LIN {X 0,Y 566.232,Z 349.956,A -85,B 0,C 180,E1 -2396.899,E2 -2396.899} C_VEL
LIN {X 0,Y 566.183,Z 349.956,A -85,B 0,C 180,E1 -2399.407,E2 -2399.407} C_VEL
LIN {X 0,Y 566.232,Z 349.955,A -85,B 0,C 180,E1 -2401.859,E2 -2401.859} C_VEL
LIN {X 0,Y 566.218,Z 349.953,A -85,B 0,C 180,E1 -2404.251,E2 -2404.251} C_VEL
LIN {X 0,Y 566.176,Z 349.96,A -85,B 0,C 180,E1 -2406.718,E2 -2406.718} C_VEL
LIN {X 0,Y 566.215,Z 349.952,A -85,B 0,C 180,E1 -2409.663,E2 -2409.663} C_VEL
LIN {X 0,Y 566.207,Z 349.954,A -85,B 0,C 180,E1 -2412.669,E2 -2412.669} C_VEL
LIN {X 0,Y 566.238,Z 349.953,A -85,B 0,C 180,E1 -2415.627,E2 -2415.627} C_VEL
LIN {X 0,Y 566.239,Z 349.956,A -85,B 0,C 180,E1 -2418.675,E2 -2418.675} C_VEL
LIN {X 0,Y 566.23,Z 349.95,A -85,B 0,C 180,E1 -2421.434,E2 -2421.434} C_VEL
LIN {X 0,Y 566.266,Z 349.947,A -85,B 0,C 180,E1 -2424.302,E2 -2424.302} C_VEL
LIN {X 0,Y 566.287,Z 349.944,A -85,B 0,C 180,E1 -2427.866,E2 -2427.866} C_VEL
LIN {X 0,Y 566.306,Z 349.944,A -85,B 0,C 180,E1 -2430.711,E2 -2430.711} C_VEL
LIN {X 0,Y 566.272,Z 349.945,A -85,B 0,C 180,E1 -2432.846,E2 -2432.846} C_VEL
LIN {X 0,Y 566.268,Z 349.949,A -85,B 0,C 180,E1 -2435.698,E2 -2435.698} C_VEL
LIN {X 0,Y 566.231,Z 349.955,A -85,B 0,C 180,E1 -2438.566,E2 -2438.566} C_VEL
LIN {X 0,Y 566.246,Z 349.949,A -85,B 0,C 180,E1 -2441.454,E2 -2441.454} C_VEL
LIN {X 0,Y 566.238,Z 349.949,A -85,B 0,C 180,E1 -2444.507,E2 -2444.507} C_VEL
LIN {X 0,Y 566.204,Z 349.958,A -85,B 0,C 180,E1 -2447.332,E2 -2447.332} C_VEL
LIN {X 0,Y 566.213,Z 349.959,A -85,B 0,C 180,E1 -2450.337,E2 -2450.337} C_VEL
LIN {X 0,Y 566.177,Z 349.958,A -85,B 0,C 180,E1 -2453.282,E2 -2453.282} C_VEL
LIN {X 0,Y 566.218,Z 349.955,A -85,B 0,C 180,E1 -2455.749,E2 -2455.749} C_VEL
LIN {X 0,Y 566.207,Z 349.954,A -85,B 0,C 180,E1 -2458.202,E2 -2458.202} C_VEL
LIN {X 0,Y 566.194,Z 349.956,A -85,B 0,C 180,E1 -2461.076,E2 -2461.076} C_VEL
LIN {X 0,Y 566.215,Z 349.959,A -85,B 0,C 180,E1 -2463.734,E2 -2463.734} C_VEL
LIN {X 0,Y 566.203,Z 349.954,A -85,B 0,C 180,E1 -2466.57,E2 -2466.57} C_VEL
LIN {X 0,Y 566.219,Z 349.952,A -85,B 0,C 180,E1 -2469.686,E2 -2469.686} C_VEL
LIN {X 0,Y 566.218,Z 349.958,A -85,B 0,C 180,E1 -2472.087,E2 -2472.087} C_VEL
LIN {X 0,Y 566.172,Z 349.959,A -85,B 0,C 180,E1 -2475.036,E2 -2475.036} C_VEL
LIN {X 0,Y 566.192,Z 349.955,A -85,B 0,C 180,E1 -2477.91,E2 -2477.91} C_VEL
LIN {X 0,Y 566.226,Z 349.955,A -85,B 0,C 180,E1 -2480.727,E2 -2480.727} C_VEL
LIN {X 0,Y 566.211,Z 349.959,A -85,B 0,C 180,E1 -2483.785,E2 -2483.785} C_VEL
LIN {X 0,Y 566.216,Z 349.952,A -85,B 0,C 180,E1 -2486.266,E2 -2486.266} C_VEL
LIN {X 0,Y 566.198,Z 349.961,A -85,B 0,C 180,E1 -2488.923,E2 -2488.923} C_VEL
LIN {X 0,Y 566.253,Z 350.125,A -85,B 0,C 180,E1 -2490.234,E2 -2490.234} C_VEL
LIN {X 0,Y 566.179,Z 357.411,A -85,B 0,C 180,E1 -2493.347,E2 -2493.347} C_VEL
LIN {X 0,Y 566.127,Z 363.027,A -85,B 0,C 180,E1 -2495.816,E2 -2495.816} C_VEL
LIN {X 0,Y 566.063,Z 370.064,A -85,B 0,C 180,E1 -2498.897,E2 -2498.897} C_VEL
LIN {X 0,Y 566.005,Z 377.154,A -85,B 0,C 180,E1 -2501.915,E2 -2501.915} C_VEL
LIN {X 0,Y 565.961,Z 382.566,A -85,B 0,C 180,E1 -2504.146,E2 -2504.146} C_VEL
LIN {X 0,Y 565.962,Z 387.979,A -85,B 0,C 180,E1 -2506.353,E2 -2506.353} C_VEL
LIN {X 0,Y 565.925,Z 395.195,A -85,B 0,C 180,E1 -2509.264,E2 -2509.264} C_VEL
LIN {X 0,Y 565.928,Z 403.709,A -85,B 0,C 180,E1 -2512.665,E2 -2512.665} C_VEL
LIN {X 0,Y 566.231,Z 412.154,A -85,B 0,C 180,E1 -2512.959,E2 -2512.959} C_VEL
LIN {X 0,Y 566.146,Z 420.811,A -85,B 0,C 180,E1 -2513.393,E2 -2513.393} C_VEL
LIN {X 0,Y 566.094,Z 429.047,A -85,B 0,C 180,E1 -2513.942,E2 -2513.942} C_VEL
LIN {X 0,Y 566.027,Z 437.057,A -85,B 0,C 180,E1 -2514.657,E2 -2514.657} C_VEL
LIN {X 0,Y 566.028,Z 443.23,A -85,B 0,C 180,E1 -2515.371,E2 -2515.371} C_VEL
LIN {X 0,Y 566.012,Z 448.087,A -85,B 0,C 180,E1 -2516.084,E2 -2516.084} C_VEL
LIN {X 0,Y 565.934,Z 451.834,A -85,B 0,C 180,E1 -2516.796,E2 -2516.796} C_VEL
LIN {X 0,Y 565.855,Z 455.839,A -85,B 0,C 180,E1 -2517.865,E2 -2517.865} C_VEL
LIN {X 0,Y 565.848,Z 457.579,A -85,B 0,C 180,E1 -2518.577,E2 -2518.577} C_VEL
LIN {X 0,Y 565.842,Z 458.621,A -85,B 0,C 180,E1 -2519.288,E2 -2519.288} C_VEL
LIN {X 0,Y 565.839,Z 458.996,A -85,B 0,C 180,E1 -2520,E2 -2520} C_VEL
LIN {X 0,Y 565.841,Z 458.711,A -85,B 0,C 180,E1 -2520.712,E2 -2520.712} C_VEL
LIN {X 0,Y 565.848,Z 457.761,A -85,B 0,C 180,E1 -2521.423,E2 -2521.423} C_VEL
LIN {X 0,Y 565.854,Z 456.12,A -85,B 0,C 180,E1 -2522.135,E2 -2522.135} C_VEL
LIN {X 0,Y 565.893,Z 453.732,A -85,B 0,C 180,E1 -2522.847,E2 -2522.847} C_VEL
LIN {X 0,Y 565.991,Z 448.601,A -85,B 0,C 180,E1 -2523.916,E2 -2523.916} C_VEL
LIN {X 0,Y 566.035,Z 442.528,A -85,B 0,C 180,E1 -2524.808,E2 -2524.808} C_VEL
LIN {X 0,Y 565.983,Z 436.212,A -85,B 0,C 180,E1 -2525.522,E2 -2525.522} C_VEL
LIN {X 0,Y 566.114,Z 429.057,A -85,B 0,C 180,E1 -2526.147,E2 -2526.147} C_VEL
LIN {X 0,Y 566.115,Z 420.691,A -85,B 0,C 180,E1 -2526.705,E2 -2526.705} C_VEL
LIN {X 0,Y 566.246,Z 411.008,A -85,B 0,C 180,E1 -2527.174,E2 -2527.174} C_VEL
LIN {X 0,Y 565.909,Z 403.653,A -85,B 0,C 180,E1 -2527.448,E2 -2527.448} C_VEL
LIN {X 0,Y 565.924,Z 395.42,A -85,B 0,C 180,E1 -2530.736,E2 -2530.736} C_VEL
LIN {X 0,Y 565.943,Z 388.201,A -85,B 0,C 180,E1 -2533.647,E2 -2533.647} C_VEL
LIN {X 0,Y 565.976,Z 380.981,A -85,B 0,C 180,E1 -2536.595,E2 -2536.595} C_VEL
LIN {X 0,Y 566.022,Z 374.496,A -85,B 0,C 180,E1 -2539.325,E2 -2539.325} C_VEL
LIN {X 0,Y 566.094,Z 368.863,A -85,B 0,C 180,E1 -2541.867,E2 -2541.867} C_VEL
LIN {X 0,Y 566.164,Z 363.641,A -85,B 0,C 180,E1 -2544.182,E2 -2544.182} C_VEL
LIN {X 0,Y 566.204,Z 357.666,A -85,B 0,C 180,E1 -2546.658,E2 -2546.658} C_VEL
LIN {X 0,Y 566.274,Z 349.951,A -85,B 0,C 180,E1 -2549.97,E2 -2549.97} C_VEL
LIN {X 0,Y 566.224,Z 349.956,A -85,B 0,C 180,E1 -2553.102,E2 -2553.102} C_VEL
LIN {X 0,Y 566.167,Z 349.964,A -85,B 0,C 180,E1 -2555.692,E2 -2555.692} C_VEL
LIN {X 0,Y 566.22,Z 349.956,A -85,B 0,C 180,E1 -2558.559,E2 -2558.559} C_VEL
LIN {X 0,Y 566.216,Z 349.959,A -85,B 0,C 180,E1 -2561.136,E2 -2561.136} C_VEL
LIN {X 0,Y 566.205,Z 349.959,A -85,B 0,C 180,E1 -2564.035,E2 -2564.035} C_VEL
LIN {X 0,Y 566.209,Z 349.958,A -85,B 0,C 180,E1 -2567.082,E2 -2567.082} C_VEL
LIN {X 0,Y 566.21,Z 349.958,A -85,B 0,C 180,E1 -2569.801,E2 -2569.801} C_VEL
LIN {X 0,Y 566.201,Z 349.961,A -85,B 0,C 180,E1 -2572.599,E2 -2572.599} C_VEL
LIN {X 0,Y 566.203,Z 349.959,A -85,B 0,C 180,E1 -2575.181,E2 -2575.181} C_VEL
LIN {X 0,Y 566.236,Z 349.957,A -85,B 0,C 180,E1 -2577.744,E2 -2577.744} C_VEL
LIN {X 0,Y 566.232,Z 350.075,A -85,B 0,C 180,E1 -2580.922,E2 -2580.922} C_VEL
LIN {X 0,Y 567.515,Z 356.097,A -85,B 0,C 180,E1 -2582.128,E2 -2582.128} C_VEL
LIN {X 0,Y 567.256,Z 368.377,A -85,B 0,C 180,E1 -2584.302,E2 -2584.302} C_VEL
LIN {X 0,Y 567.027,Z 381.516,A -85,B 0,C 180,E1 -2586.519,E2 -2586.519} C_VEL
LIN {X 0,Y 566.812,Z 397.208,A -85,B 0,C 180,E1 -2589.116,E2 -2589.116} C_VEL
LIN {X 0,Y 566.567,Z 414.516,A -85,B 0,C 180,E1 -2591.934,E2 -2591.934} C_VEL
LIN {X 0,Y 566.392,Z 432.979,A -85,B 0,C 180,E1 -2594.896,E2 -2594.896} C_VEL
LIN {X 0,Y 566.217,Z 447.98,A -85,B 0,C 180,E1 -2597.272,E2 -2597.272} C_VEL
LIN {X 0,Y 566.942,Z 453.599,A -85,B 0,C 180,E1 -2597.38,E2 -2597.38} C_VEL
LIN {X 0,Y 566.899,Z 466.689,A -85,B 0,C 180,E1 -2597.674,E2 -2597.674} C_VEL
LIN {X 0,Y 566.748,Z 479.914,A -85,B 0,C 180,E1 -2598.13,E2 -2598.13} C_VEL
LIN {X 0,Y 566.61,Z 492.108,A -85,B 0,C 180,E1 -2598.705,E2 -2598.705} C_VEL
LIN {X 0,Y 566.485,Z 502.907,A -85,B 0,C 180,E1 -2599.365,E2 -2599.365} C_VEL
LIN {X 0,Y 566.339,Z 513.539,A -85,B 0,C 180,E1 -2600.175,E2 -2600.175} C_VEL
LIN {X 0,Y 566.207,Z 523.111,A -85,B 0,C 180,E1 -2601.074,E2 -2601.074} C_VEL
LIN {X 0,Y 566.112,Z 530.959,A -85,B 0,C 180,E1 -2601.971,E2 -2601.971} C_VEL
LIN {X 0,Y 566.001,Z 538.621,A -85,B 0,C 180,E1 -2603.046,E2 -2603.046} C_VEL
LIN {X 0,Y 566.004,Z 545.679,A -85,B 0,C 180,E1 -2604.299,E2 -2604.299} C_VEL
LIN {X 0,Y 565.933,Z 550.372,A -85,B 0,C 180,E1 -2605.37,E2 -2605.37} C_VEL
LIN {X 0,Y 565.927,Z 553.957,A -85,B 0,C 180,E1 -2606.44,E2 -2606.44} C_VEL
LIN {X 0,Y 565.878,Z 555.808,A -85,B 0,C 180,E1 -2607.152,E2 -2607.152} C_VEL
LIN {X 0,Y 565.846,Z 558.185,A -85,B 0,C 180,E1 -2608.576,E2 -2608.576} C_VEL
LIN {X 0,Y 565.839,Z 559,A -85,B 0,C 180,E1 -2610,E2 -2610} C_VEL
LIN {X 0,Y 565.846,Z 558.186,A -85,B 0,C 180,E1 -2611.423,E2 -2611.423} C_VEL
LIN {X 0,Y 565.878,Z 555.81,A -85,B 0,C 180,E1 -2612.847,E2 -2612.847} C_VEL
LIN {X 0,Y 565.926,Z 552.897,A -85,B 0,C 180,E1 -2613.916,E2 -2613.916} C_VEL
LIN {X 0,Y 565.878,Z 548.95,A -85,B 0,C 180,E1 -2614.987,E2 -2614.987} C_VEL
LIN {X 0,Y 566.002,Z 543.868,A -85,B 0,C 180,E1 -2616.058,E2 -2616.058} C_VEL
LIN {X 0,Y 566.04,Z 537.468,A -85,B 0,C 180,E1 -2617.132,E2 -2617.132} C_VEL
LIN {X 0,Y 566.133,Z 529.48,A -85,B 0,C 180,E1 -2618.208,E2 -2618.208} C_VEL
LIN {X 0,Y 566.229,Z 521.336,A -85,B 0,C 180,E1 -2619.105,E2 -2619.105} C_VEL
LIN {X 0,Y 566.35,Z 511.402,A -85,B 0,C 180,E1 -2620.005,E2 -2620.005} C_VEL
LIN {X 0,Y 566.524,Z 500.284,A -85,B 0,C 180,E1 -2620.808,E2 -2620.808} C_VEL
LIN {X 0,Y 566.66,Z 489.178,A -85,B 0,C 180,E1 -2621.446,E2 -2621.446} C_VEL
LIN {X 0,Y 566.746,Z 476.986,A -85,B 0,C 180,E1 -2621.988,E2 -2621.988} C_VEL
LIN {X 0,Y 566.887,Z 464.18,A -85,B 0,C 180,E1 -2622.394,E2 -2622.394} C_VEL
LIN {X 0,Y 566.827,Z 452.111,A -85,B 0,C 180,E1 -2622.645,E2 -2622.645} C_VEL
LIN {X 0,Y 566.216,Z 447.982,A -85,B 0,C 180,E1 -2622.728,E2 -2622.728} C_VEL
LIN {X 0,Y 566.399,Z 431.827,A -85,B 0,C 180,E1 -2625.288,E2 -2625.288} C_VEL
LIN {X 0,Y 566.568,Z 414.518,A -85,B 0,C 180,E1 -2628.066,E2 -2628.066} C_VEL
LIN {X 0,Y 566.791,Z 398.363,A -85,B 0,C 180,E1 -2630.695,E2 -2630.695} C_VEL
LIN {X 0,Y 567.037,Z 381.524,A -85,B 0,C 180,E1 -2633.483,E2 -2633.483} C_VEL
LIN {X 0,Y 567.381,Z 363.879,A -85,B 0,C 180,E1 -2636.482,E2 -2636.482} C_VEL
LIN {X 0,Y 567.421,Z 355.866,A -85,B 0,C 180,E1 -2637.876,E2 -2637.876} C_VEL
LIN {X 0,Y 566.23,Z 349.956,A -85,B 0,C 180,E1 -2639.002,E2 -2639.002} C_VEL
LIN {X 0,Y 566.235,Z 349.953,A -85,B 0,C 180,E1 -2642.256,E2 -2642.256} C_VEL
LIN {X 0,Y 566.184,Z 349.962,A -85,B 0,C 180,E1 -2644.99,E2 -2644.99} C_VEL
LIN {X 0,Y 566.198,Z 349.955,A -85,B 0,C 180,E1 -2647.461,E2 -2647.461} C_VEL
LIN {X 0,Y 566.209,Z 349.96,A -85,B 0,C 180,E1 -2650.199,E2 -2650.199} C_VEL
LIN {X 0,Y 566.208,Z 349.955,A -85,B 0,C 180,E1 -2653.054,E2 -2653.054} C_VEL
LIN {X 0,Y 566.204,Z 349.954,A -85,B 0,C 180,E1 -2656.048,E2 -2656.048} C_VEL
LIN {X 0,Y 566.222,Z 349.951,A -85,B 0,C 180,E1 -2659.212,E2 -2659.212} C_VEL
LIN {X 0,Y 566.192,Z 349.959,A -85,B 0,C 180,E1 -2661.637,E2 -2661.637} C_VEL
LIN {X 0,Y 566.199,Z 349.955,A -85,B 0,C 180,E1 -2664.31,E2 -2664.31} C_VEL
LIN {X 0,Y 566.222,Z 349.957,A -85,B 0,C 180,E1 -2666.898,E2 -2666.898} C_VEL
LIN {X 0,Y 566.19,Z 349.955,A -85,B 0,C 180,E1 -2669.408,E2 -2669.408} C_VEL
LIN {X 0,Y 566.231,Z 349.957,A -85,B 0,C 180,E1 -2671.858,E2 -2671.858} C_VEL
LIN {X 0,Y 566.215,Z 349.953,A -85,B 0,C 180,E1 -2674.251,E2 -2674.251} C_VEL
LIN {X 0,Y 566.171,Z 349.963,A -85,B 0,C 180,E1 -2676.719,E2 -2676.719} C_VEL
LIN {X 0,Y 566.215,Z 349.953,A -85,B 0,C 180,E1 -2679.663,E2 -2679.663} C_VEL
LIN {X 0,Y 566.201,Z 349.954,A -85,B 0,C 180,E1 -2682.668,E2 -2682.668} C_VEL
LIN {X 0,Y 566.237,Z 349.952,A -85,B 0,C 180,E1 -2685.627,E2 -2685.627} C_VEL
LIN {X 0,Y 566.237,Z 349.955,A -85,B 0,C 180,E1 -2688.675,E2 -2688.675} C_VEL
LIN {X 0,Y 566.23,Z 349.952,A -85,B 0,C 180,E1 -2691.434,E2 -2691.434} C_VEL
LIN {X 0,Y 566.258,Z 349.947,A -85,B 0,C 180,E1 -2694.302,E2 -2694.302} C_VEL
LIN {X 0,Y 566.278,Z 349.945,A -85,B 0,C 180,E1 -2697.866,E2 -2697.866} C_VEL
LIN {X 0,Y 566.305,Z 349.943,A -85,B 0,C 180,E1 -2700.711,E2 -2700.711} C_VEL
LIN {X 0,Y 566.275,Z 349.945,A -85,B 0,C 180,E1 -2702.846,E2 -2702.846} C_VEL
LIN {X 0,Y 566.261,Z 349.948,A -85,B 0,C 180,E1 -2705.698,E2 -2705.698} C_VEL
LIN {X 0,Y 566.236,Z 349.956,A -85,B 0,C 180,E1 -2708.566,E2 -2708.566} C_VEL
LIN {X 0,Y 566.244,Z 349.95,A -85,B 0,C 180,E1 -2711.454,E2 -2711.454} C_VEL
LIN {X 0,Y 566.236,Z 349.949,A -85,B 0,C 180,E1 -2714.507,E2 -2714.507} C_VEL
LIN {X 0,Y 566.202,Z 349.956,A -85,B 0,C 180,E1 -2717.332,E2 -2717.332} C_VEL
LIN {X 0,Y 566.216,Z 349.959,A -85,B 0,C 180,E1 -2720.337,E2 -2720.337} C_VEL
LIN {X 0,Y 566.191,Z 349.96,A -85,B 0,C 180,E1 -2723.404,E2 -2723.404} C_VEL
LIN {X 0,Y 566.215,Z 349.953,A -85,B 0,C 180,E1 -2725.749,E2 -2725.749} C_VEL
LIN {X 0,Y 566.205,Z 349.954,A -85,B 0,C 180,E1 -2727.483,E2 -2727.483} C_VEL
LIN {X 0,Y 565.525,Z 350.04,A -85,B 0,C 180,E1 -2728.077,E2 -2728.077} C_VEL
LIN {X 0,Y 562.659,Z 350.397,A -85,B 0,C 180,E1 -2729.04,E2 -2729.04} C_VEL
LIN {X 0,Y 560.249,Z 350.699,A -85,B 0,C 180,E1 -2729.816,E2 -2729.816} C_VEL
LIN {X 0,Y 559.222,Z 350.829,A -85,B 0,C 180,E1 -2730.414,E2 -2730.414} C_VEL
LIN {X 0,Y 559.141,Z 350.835,A -85,B 0,C 180,E1 -2730.617,E2 -2730.617} C_VEL
LIN {X 0,Y 559.167,Z 350.837,A -85,B 0,C 180,E1 -2733.575,E2 -2733.575} C_VEL
LIN {X 0,Y 559.16,Z 350.832,A -85,B 0,C 180,E1 -2736.447,E2 -2736.447} C_VEL
LIN {X 0,Y 559.18,Z 350.832,A -85,B 0,C 180,E1 -2738.934,E2 -2738.934} C_VEL
LIN {X 0,Y 559.193,Z 350.831,A -85,B 0,C 180,E1 -2741.768,E2 -2741.768} C_VEL
LIN {X 0,Y 559.142,Z 350.834,A -85,B 0,C 180,E1 -2744.739,E2 -2744.739} C_VEL
LIN {X 0,Y 559.167,Z 350.833,A -85,B 0,C 180,E1 -2747.257,E2 -2747.257} C_VEL
LIN {X 0,Y 559.182,Z 350.832,A -85,B 0,C 180,E1 -2750.135,E2 -2750.135} C_VEL
LIN {X 0,Y 559.143,Z 350.834,A -85,B 0,C 180,E1 -2752.892,E2 -2752.892} C_VEL
LIN {X 0,Y 559.169,Z 350.831,A -85,B 0,C 180,E1 -2756.051,E2 -2756.051} C_VEL
LIN {X 0,Y 559.158,Z 350.834,A -85,B 0,C 180,E1 -2758.981,E2 -2758.981} C_VEL
LIN {X 0,Y 559.173,Z 350.831,A -85,B 0,C 180,E1 -2761.619,E2 -2761.619} C_VEL
LIN {X 0,Y 559.185,Z 350.833,A -85,B 0,C 180,E1 -2763.903,E2 -2763.903} C_VEL
LIN {X 0,Y 559.145,Z 350.835,A -85,B 0,C 180,E1 -2766.571,E2 -2766.571} C_VEL
LIN {X 0,Y 559.182,Z 350.828,A -85,B 0,C 180,E1 -2769.396,E2 -2769.396} C_VEL
LIN {X 0,Y 559.154,Z 350.834,A -85,B 0,C 180,E1 -2771.686,E2 -2771.686} C_VEL
LIN {X 0,Y 559.171,Z 350.834,A -85,B 0,C 180,E1 -2773.948,E2 -2773.948} C_VEL
LIN {X 0,Y 559.176,Z 350.83,A -85,B 0,C 180,E1 -2776.184,E2 -2776.184} C_VEL
LIN {X 0,Y 559.199,Z 350.828,A -85,B 0,C 180,E1 -2779.134,E2 -2779.134} C_VEL
LIN {X 0,Y 559.207,Z 350.832,A -85,B 0,C 180,E1 -2782.054,E2 -2782.054} C_VEL
LIN {X 0,Y 559.26,Z 350.821,A -85,B 0,C 180,E1 -2784.954,E2 -2784.954} C_VEL
LIN {X 0,Y 559.258,Z 350.819,A -85,B 0,C 180,E1 -2787.84,E2 -2787.84} C_VEL
LIN {X 0,Y 559.276,Z 350.819,A -85,B 0,C 180,E1 -2790.72,E2 -2790.72} C_VEL
LIN {X 0,Y 559.239,Z 350.821,A -85,B 0,C 180,E1 -2792.882,E2 -2792.882} C_VEL
LIN {X 0,Y 559.236,Z 350.824,A -85,B 0,C 180,E1 -2795.77,E2 -2795.77} C_VEL
LIN {X 0,Y 559.19,Z 350.833,A -85,B 0,C 180,E1 -2798.674,E2 -2798.674} C_VEL
LIN {X 0,Y 559.209,Z 350.826,A -85,B 0,C 180,E1 -2801.601,E2 -2801.601} C_VEL
LIN {X 0,Y 559.204,Z 350.825,A -85,B 0,C 180,E1 -2804.596,E2 -2804.596} C_VEL
LIN {X 0,Y 559.163,Z 350.833,A -85,B 0,C 180,E1 -2807.557,E2 -2807.557} C_VEL
LIN {X 0,Y 559.171,Z 350.831,A -85,B 0,C 180,E1 -2809.838,E2 -2809.838} C_VEL
LIN {X 0,Y 559.146,Z 350.839,A -85,B 0,C 180,E1 -2812.153,E2 -2812.153} C_VEL
LIN {X 0,Y 559.18,Z 350.833,A -85,B 0,C 180,E1 -2815.298,E2 -2815.298} C_VEL
LIN {X 0,Y 559.185,Z 350.829,A -85,B 0,C 180,E1 -2817.712,E2 -2817.712} C_VEL
LIN {X 0,Y 559.157,Z 350.835,A -85,B 0,C 180,E1 -2820.183,E2 -2820.183} C_VEL
LIN {X 0,Y 559.179,Z 350.83,A -85,B 0,C 180,E1 -2822.714,E2 -2822.714} C_VEL
LIN {X 0,Y 559.131,Z 350.84,A -85,B 0,C 180,E1 -2825.324,E2 -2825.324} C_VEL
LIN {X 0,Y 559.137,Z 350.834,A -85,B 0,C 180,E1 -2828.018,E2 -2828.018} C_VEL
LIN {X 0,Y 559.163,Z 350.834,A -85,B 0,C 180,E1 -2830.812,E2 -2830.812} C_VEL
LIN {X 0,Y 559.167,Z 350.837,A -85,B 0,C 180,E1 -2833.732,E2 -2833.732} C_VEL
LIN {X 0,Y 559.148,Z 350.835,A -85,B 0,C 180,E1 -2836.804,E2 -2836.804} C_VEL
LIN {X 0,Y 559.159,Z 350.834,A -85,B 0,C 180,E1 -2839.188,E2 -2839.188} C_VEL
LIN {X 0,Y 559.139,Z 350.839,A -85,B 0,C 180,E1 -2841.983,E2 -2841.983} C_VEL
LIN {X 0,Y 559.152,Z 350.833,A -85,B 0,C 180,E1 -2844.785,E2 -2844.785} C_VEL
LIN {X 0,Y 559.16,Z 350.836,A -85,B 0,C 180,E1 -2847.364,E2 -2847.364} C_VEL
LIN {X 0,Y 559.221,Z 350.98,A -85,B 0,C 180,E1 -2850.205,E2 -2850.205} C_VEL
LIN {X 0,Y 559.119,Z 357.885,A -85,B 0,C 180,E1 -2853.184,E2 -2853.184} C_VEL
LIN {X 0,Y 559.069,Z 363.146,A -85,B 0,C 180,E1 -2855.491,E2 -2855.491} C_VEL
LIN {X 0,Y 558.999,Z 369.897,A -85,B 0,C 180,E1 -2858.492,E2 -2858.492} C_VEL
LIN {X 0,Y 558.955,Z 375.475,A -85,B 0,C 180,E1 -2860.919,E2 -2860.919} C_VEL
LIN {X 0,Y 558.917,Z 380.783,A -85,B 0,C 180,E1 -2863.189,E2 -2863.189} C_VEL
LIN {X 0,Y 558.867,Z 387.98,A -85,B 0,C 180,E1 -2866.176,E2 -2866.176} C_VEL
LIN {X 0,Y 558.845,Z 395.197,A -85,B 0,C 180,E1 -2869.127,E2 -2869.127} C_VEL
LIN {X 0,Y 558.824,Z 403.723,A -85,B 0,C 180,E1 -2872.571,E2 -2872.571} C_VEL
LIN {X 0,Y 559.198,Z 412.375,A -85,B 0,C 180,E1 -2872.879,E2 -2872.879} C_VEL
LIN {X 0,Y 559.091,Z 421.265,A -85,B 0,C 180,E1 -2873.336,E2 -2873.336} C_VEL
LIN {X 0,Y 559.054,Z 429.057,A -85,B 0,C 180,E1 -2873.866,E2 -2873.866} C_VEL
LIN {X 0,Y 558.934,Z 437.062,A -85,B 0,C 180,E1 -2874.589,E2 -2874.589} C_VEL
LIN {X 0,Y 558.967,Z 443.233,A -85,B 0,C 180,E1 -2875.312,E2 -2875.312} C_VEL
LIN {X 0,Y 558.919,Z 448.091,A -85,B 0,C 180,E1 -2876.034,E2 -2876.034} C_VEL
LIN {X 0,Y 558.859,Z 451.836,A -85,B 0,C 180,E1 -2876.756,E2 -2876.756} C_VEL
LIN {X 0,Y 558.763,Z 455.841,A -85,B 0,C 180,E1 -2877.838,E2 -2877.838} C_VEL
LIN {X 0,Y 558.748,Z 457.581,A -85,B 0,C 180,E1 -2878.558,E2 -2878.558} C_VEL
LIN {X 0,Y 558.742,Z 458.622,A -85,B 0,C 180,E1 -2879.279,E2 -2879.279} C_VEL
LIN {X 0,Y 558.74,Z 458.996,A -85,B 0,C 180,E1 -2880,E2 -2880} C_VEL
LIN {X 0,Y 558.742,Z 458.71,A -85,B 0,C 180,E1 -2880.721,E2 -2880.721} C_VEL
LIN {X 0,Y 558.748,Z 457.76,A -85,B 0,C 180,E1 -2881.441,E2 -2881.441} C_VEL
LIN {X 0,Y 558.762,Z 456.118,A -85,B 0,C 180,E1 -2882.162,E2 -2882.162} C_VEL
LIN {X 0,Y 558.816,Z 453.73,A -85,B 0,C 180,E1 -2882.884,E2 -2882.884} C_VEL
LIN {X 0,Y 558.889,Z 448.598,A -85,B 0,C 180,E1 -2883.966,E2 -2883.966} C_VEL
LIN {X 0,Y 558.961,Z 442.523,A -85,B 0,C 180,E1 -2884.869,E2 -2884.869} C_VEL
LIN {X 0,Y 558.924,Z 436.206,A -85,B 0,C 180,E1 -2885.592,E2 -2885.592} C_VEL
LIN {X 0,Y 559.061,Z 429.051,A -85,B 0,C 180,E1 -2886.225,E2 -2886.225} C_VEL
LIN {X 0,Y 559.081,Z 421.473,A -85,B 0,C 180,E1 -2886.742,E2 -2886.742} C_VEL
LIN {X 0,Y 559.199,Z 412.166,A -85,B 0,C 180,E1 -2887.22,E2 -2887.22} C_VEL
LIN {X 0,Y 558.8,Z 403.652,A -85,B 0,C 180,E1 -2887.543,E2 -2887.543} C_VEL
LIN {X 0,Y 558.844,Z 395.418,A -85,B 0,C 180,E1 -2890.873,E2 -2890.873} C_VEL
LIN {X 0,Y 558.852,Z 388.199,A -85,B 0,C 180,E1 -2893.824,E2 -2893.824} C_VEL
LIN {X 0,Y 558.908,Z 381.045,A -85,B 0,C 180,E1 -2896.811,E2 -2896.811} C_VEL
LIN {X 0,Y 558.997,Z 375.13,A -85,B 0,C 180,E1 -2899.448,E2 -2899.448} C_VEL
LIN {X 0,Y 559.065,Z 369.217,A -85,B 0,C 180,E1 -2902.156,E2 -2902.156} C_VEL
LIN {X 0,Y 559.142,Z 362.057,A -85,B 0,C 180,E1 -2905.178,E2 -2905.178} C_VEL
LIN {X 0,Y 559.157,Z 356.253,A -85,B 0,C 180,E1 -2907.714,E2 -2907.714} C_VEL
LIN {X 0,Y 559.252,Z 350.826,A -85,B 0,C 180,E1 -2910.036,E2 -2910.036} C_VEL
LIN {X 0,Y 559.16,Z 350.838,A -85,B 0,C 180,E1 -2912.715,E2 -2912.715} C_VEL
LIN {X 0,Y 559.132,Z 350.839,A -85,B 0,C 180,E1 -2915.324,E2 -2915.324} C_VEL
LIN {X 0,Y 559.139,Z 350.84,A -85,B 0,C 180,E1 -2918.017,E2 -2918.017} C_VEL
LIN {X 0,Y 559.181,Z 350.834,A -85,B 0,C 180,E1 -2920.81,E2 -2920.81} C_VEL
LIN {X 0,Y 559.167,Z 350.835,A -85,B 0,C 180,E1 -2923.732,E2 -2923.732} C_VEL
LIN {X 0,Y 559.172,Z 350.834,A -85,B 0,C 180,E1 -2926.801,E2 -2926.801} C_VEL
LIN {X 0,Y 559.163,Z 350.836,A -85,B 0,C 180,E1 -2929.188,E2 -2929.188} C_VEL
LIN {X 0,Y 559.134,Z 350.839,A -85,B 0,C 180,E1 -2931.982,E2 -2931.982} C_VEL
LIN {X 0,Y 559.136,Z 350.841,A -85,B 0,C 180,E1 -2934.787,E2 -2934.787} C_VEL
LIN {X 0,Y 559.178,Z 350.835,A -85,B 0,C 180,E1 -2937.361,E2 -2937.361} C_VEL
LIN {X 0,Y 559.196,Z 350.833,A -85,B 0,C 180,E1 -2940.484,E2 -2940.484} C_VEL
LIN {X 0,Y 559.217,Z 351.017,A -85,B 0,C 180,E1 -2940.65,E2 -2940.65} C_VEL
LIN {X 0,Y 560.68,Z 358.415,A -85,B 0,C 180,E1 -2942.165,E2 -2942.165} C_VEL
LIN {X 0,Y 560.334,Z 370.412,A -85,B 0,C 180,E1 -2944.328,E2 -2944.328} C_VEL
LIN {X 0,Y 560.057,Z 382.721,A -85,B 0,C 180,E1 -2946.456,E2 -2946.456} C_VEL
LIN {X 0,Y 559.877,Z 398.362,A -85,B 0,C 180,E1 -2949.037,E2 -2949.037} C_VEL
LIN {X 0,Y 559.576,Z 416.824,A -85,B 0,C 180,E1 -2952.079,E2 -2952.079} C_VEL
LIN {X 0,Y 559.357,Z 434.248,A -85,B 0,C 180,E1 -2954.906,E2 -2954.906} C_VEL
LIN {X 0,Y 559.207,Z 448.188,A -85,B 0,C 180,E1 -2957.121,E2 -2957.121} C_VEL
LIN {X 0,Y 560.033,Z 454.937,A -85,B 0,C 180,E1 -2957.244,E2 -2957.244} C_VEL
LIN {X 0,Y 559.948,Z 468.212,A -85,B 0,C 180,E1 -2957.565,E2 -2957.565} C_VEL
LIN {X 0,Y 559.805,Z 481.149,A -85,B 0,C 180,E1 -2958.031,E2 -2958.031} C_VEL
LIN {X 0,Y 559.626,Z 492.864,A -85,B 0,C 180,E1 -2958.606,E2 -2958.606} C_VEL
LIN {X 0,Y 559.478,Z 504.197,A -85,B 0,C 180,E1 -2959.322,E2 -2959.322} C_VEL
LIN {X 0,Y 559.308,Z 514.6,A -85,B 0,C 180,E1 -2960.142,E2 -2960.142} C_VEL
LIN {X 0,Y 559.162,Z 523.111,A -85,B 0,C 180,E1 -2960.961,E2 -2960.961} C_VEL
LIN {X 0,Y 559.05,Z 530.959,A -85,B 0,C 180,E1 -2961.869,E2 -2961.869} C_VEL
LIN {X 0,Y 558.943,Z 538.621,A -85,B 0,C 180,E1 -2962.958,E2 -2962.958} C_VEL
LIN {X 0,Y 558.935,Z 545.679,A -85,B 0,C 180,E1 -2964.227,E2 -2964.227} C_VEL
LIN {X 0,Y 558.826,Z 550.372,A -85,B 0,C 180,E1 -2965.311,E2 -2965.311} C_VEL
LIN {X 0,Y 558.836,Z 553.957,A -85,B 0,C 180,E1 -2966.395,E2 -2966.395} C_VEL
LIN {X 0,Y 558.799,Z 555.807,A -85,B 0,C 180,E1 -2967.116,E2 -2967.116} C_VEL
LIN {X 0,Y 558.746,Z 558.185,A -85,B 0,C 180,E1 -2968.558,E2 -2968.558} C_VEL
LIN {X 0,Y 558.74,Z 559,A -85,B 0,C 180,E1 -2970,E2 -2970} C_VEL
LIN {X 0,Y 558.746,Z 558.186,A -85,B 0,C 180,E1 -2971.441,E2 -2971.441} C_VEL
LIN {X 0,Y 558.799,Z 555.81,A -85,B 0,C 180,E1 -2972.884,E2 -2972.884} C_VEL
LIN {X 0,Y 558.843,Z 552.897,A -85,B 0,C 180,E1 -2973.966,E2 -2973.966} C_VEL
LIN {X 0,Y 558.798,Z 548.95,A -85,B 0,C 180,E1 -2975.051,E2 -2975.051} C_VEL
LIN {X 0,Y 558.919,Z 543.868,A -85,B 0,C 180,E1 -2976.135,E2 -2976.135} C_VEL
LIN {X 0,Y 558.977,Z 537.468,A -85,B 0,C 180,E1 -2977.223,E2 -2977.223} C_VEL
LIN {X 0,Y 559.099,Z 529.479,A -85,B 0,C 180,E1 -2978.312,E2 -2978.312} C_VEL
LIN {X 0,Y 559.195,Z 521.336,A -85,B 0,C 180,E1 -2979.221,E2 -2979.221} C_VEL
LIN {X 0,Y 559.36,Z 511.402,A -85,B 0,C 180,E1 -2980.131,E2 -2980.131} C_VEL
LIN {X 0,Y 559.527,Z 500.365,A -85,B 0,C 180,E1 -2980.939,E2 -2980.939} C_VEL
LIN {X 0,Y 559.703,Z 488.144,A -85,B 0,C 180,E1 -2981.644,E2 -2981.644} C_VEL
LIN {X 0,Y 559.839,Z 475.769,A -85,B 0,C 180,E1 -2982.184,E2 -2982.184} C_VEL
LIN {X 0,Y 559.963,Z 462.35,A -85,B 0,C 180,E1 -2982.596,E2 -2982.596} C_VEL
LIN {X 0,Y 559.825,Z 452.115,A -85,B 0,C 180,E1 -2982.806,E2 -2982.806} C_VEL
LIN {X 0,Y 559.219,Z 447.982,A -85,B 0,C 180,E1 -2982.89,E2 -2982.89} C_VEL
LIN {X 0,Y 559.39,Z 430.673,A -85,B 0,C 180,E1 -2985.671,E2 -2985.671} C_VEL
LIN {X 0,Y 559.615,Z 413.364,A -85,B 0,C 180,E1 -2988.488,E2 -2988.488} C_VEL
LIN {X 0,Y 559.867,Z 397.209,A -85,B 0,C 180,E1 -2991.155,E2 -2991.155} C_VEL
LIN {X 0,Y 560.121,Z 382.29,A -85,B 0,C 180,E1 -2993.673,E2 -2993.673} C_VEL
LIN {X 0,Y 560.512,Z 365.102,A -85,B 0,C 180,E1 -2996.632,E2 -2996.632} C_VEL
LIN {X 0,Y 560.509,Z 357.089,A -85,B 0,C 180,E1 -2998.047,E2 -2998.047} C_VEL
LIN {X 0,Y 559.19,Z 350.832,A -85,B 0,C 180,E1 -2999.248,E2 -2999.248} C_VEL
LIN {X 0,Y 559.169,Z 350.836,A -85,B 0,C 180,E1 -3001.862,E2 -3001.862} C_VEL
LIN {X 0,Y 559.146,Z 350.834,A -85,B 0,C 180,E1 -3004.445,E2 -3004.445} C_VEL
LIN {X 0,Y 559.143,Z 350.836,A -85,B 0,C 180,E1 -3007.108,E2 -3007.108} C_VEL
LIN {X 0,Y 559.163,Z 350.835,A -85,B 0,C 180,E1 -3009.942,E2 -3009.942} C_VEL
LIN {X 0,Y 559.166,Z 350.831,A -85,B 0,C 180,E1 -3012.743,E2 -3012.743} C_VEL
LIN {X 0,Y 559.158,Z 350.832,A -85,B 0,C 180,E1 -3015.76,E2 -3015.76} C_VEL
LIN {X 0,Y 559.168,Z 350.834,A -85,B 0,C 180,E1 -3018.23,E2 -3018.23} C_VEL
LIN {X 0,Y 559.18,Z 350.829,A -85,B 0,C 180,E1 -3021.191,E2 -3021.191} C_VEL
LIN {X 0,Y 559.164,Z 350.834,A -85,B 0,C 180,E1 -3023.791,E2 -3023.791} C_VEL
LIN {X 0,Y 559.165,Z 350.833,A -85,B 0,C 180,E1 -3026.425,E2 -3026.425} C_VEL
LIN {X 0,Y 559.165,Z 350.832,A -85,B 0,C 180,E1 -3028.981,E2 -3028.981} C_VEL
LIN {X 0,Y 559.17,Z 350.833,A -85,B 0,C 180,E1 -3031.619,E2 -3031.619} C_VEL
LIN {X 0,Y 559.183,Z 350.831,A -85,B 0,C 180,E1 -3033.903,E2 -3033.903} C_VEL
LIN {X 0,Y 559.141,Z 350.837,A -85,B 0,C 180,E1 -3036.572,E2 -3036.572} C_VEL
LIN {X 0,Y 559.182,Z 350.829,A -85,B 0,C 180,E1 -3039.395,E2 -3039.395} C_VEL
LIN {X 0,Y 559.145,Z 350.837,A -85,B 0,C 180,E1 -3041.686,E2 -3041.686} C_VEL
LIN {X 0,Y 559.169,Z 350.832,A -85,B 0,C 180,E1 -3043.948,E2 -3043.948} C_VEL
LIN {X 0,Y 559.176,Z 350.83,A -85,B 0,C 180,E1 -3046.184,E2 -3046.184} C_VEL
LIN {X 0,Y 559.197,Z 350.828,A -85,B 0,C 180,E1 -3049.134,E2 -3049.134} C_VEL
LIN {X 0,Y 559.206,Z 350.83,A -85,B 0,C 180,E1 -3052.054,E2 -3052.054} C_VEL
LIN {X 0,Y 559.257,Z 350.822,A -85,B 0,C 180,E1 -3054.953,E2 -3054.953} C_VEL
LIN {X 0,Y 559.25,Z 350.82,A -85,B 0,C 180,E1 -3057.839,E2 -3057.839} C_VEL
LIN {X 0,Y 559.275,Z 350.818,A -85,B 0,C 180,E1 -3060.72,E2 -3060.72} C_VEL
LIN {X 0,Y 559.241,Z 350.821,A -85,B 0,C 180,E1 -3062.881,E2 -3062.881} C_VEL
LIN {X 0,Y 559.23,Z 350.823,A -85,B 0,C 180,E1 -3065.77,E2 -3065.77} C_VEL
LIN {X 0,Y 559.194,Z 350.833,A -85,B 0,C 180,E1 -3068.674,E2 -3068.674} C_VEL
LIN {X 0,Y 559.208,Z 350.828,A -85,B 0,C 180,E1 -3071.6,E2 -3071.6} C_VEL
LIN {X 0,Y 559.202,Z 350.826,A -85,B 0,C 180,E1 -3074.596,E2 -3074.596} C_VEL
LIN {X 0,Y 559.162,Z 350.832,A -85,B 0,C 180,E1 -3077.557,E2 -3077.557} C_VEL
LIN {X 0,Y 559.175,Z 350.831,A -85,B 0,C 180,E1 -3079.837,E2 -3079.837} C_VEL
LIN {X 0,Y 559.143,Z 350.838,A -85,B 0,C 180,E1 -3082.153,E2 -3082.153} C_VEL
LIN {X 0,Y 559.181,Z 350.834,A -85,B 0,C 180,E1 -3085.187,E2 -3085.187} C_VEL
LIN {X 0,Y 559.159,Z 350.831,A -85,B 0,C 180,E1 -3087.713,E2 -3087.713} C_VEL
LIN {X 0,Y 559.141,Z 350.835,A -85,B 0,C 180,E1 -3090.617,E2 -3090.617} C_VEL
LIN {X 0,Y 558.481,Z 350.917,A -85,B 0,C 180,E1 -3091.219,E2 -3091.219} C_VEL
LIN {X 0,Y 555.621,Z 351.276,A -85,B 0,C 180,E1 -3092.195,E2 -3092.195} C_VEL
LIN {X 0,Y 553.211,Z 351.574,A -85,B 0,C 180,E1 -3092.981,E2 -3092.981} C_VEL
LIN {X 0,Y 552.191,Z 351.705,A -85,B 0,C 180,E1 -3093.587,E2 -3093.587} C_VEL
LIN {X 0,Y 552.116,Z 351.709,A -85,B 0,C 180,E1 -3093.793,E2 -3093.793} C_VEL
LIN {X 0,Y 552.111,Z 351.713,A -85,B 0,C 180,E1 -3096.747,E2 -3096.747} C_VEL
LIN {X 0,Y 552.134,Z 351.706,A -85,B 0,C 180,E1 -3099.527,E2 -3099.527} C_VEL
LIN {X 0,Y 552.133,Z 351.709,A -85,B 0,C 180,E1 -3102.425,E2 -3102.425} C_VEL
LIN {X 0,Y 552.102,Z 351.714,A -85,B 0,C 180,E1 -3105.563,E2 -3105.563} C_VEL
LIN {X 0,Y 552.132,Z 351.713,A -85,B 0,C 180,E1 -3108.677,E2 -3108.677} C_VEL
LIN {X 0,Y 552.12,Z 351.709,A -85,B 0,C 180,E1 -3111.411,E2 -3111.411} C_VEL
LIN {X 0,Y 552.088,Z 351.714,A -85,B 0,C 180,E1 -3114.157,E2 -3114.157} C_VEL
LIN {X 0,Y 552.126,Z 351.712,A -85,B 0,C 180,E1 -3116.815,E2 -3116.815} C_VEL
LIN {X 0,Y 552.105,Z 351.709,A -85,B 0,C 180,E1 -3119.391,E2 -3119.391} C_VEL
LIN {X 0,Y 552.129,Z 351.712,A -85,B 0,C 180,E1 -3121.903,E2 -3121.903} C_VEL
LIN {X 0,Y 552.159,Z 351.704,A -85,B 0,C 180,E1 -3124.65,E2 -3124.65} C_VEL
LIN {X 0,Y 552.096,Z 351.712,A -85,B 0,C 180,E1 -3127.549,E2 -3127.549} C_VEL
LIN {X 0,Y 552.152,Z 351.711,A -85,B 0,C 180,E1 -3130.374,E2 -3130.374} C_VEL
LIN {X 0,Y 552.16,Z 351.703,A -85,B 0,C 180,E1 -3132.978,E2 -3132.978} C_VEL
LIN {X 0,Y 552.139,Z 351.707,A -85,B 0,C 180,E1 -3136.005,E2 -3136.005} C_VEL
LIN {X 0,Y 552.167,Z 351.706,A -85,B 0,C 180,E1 -3138.994,E2 -3138.994} C_VEL
LIN {X 0,Y 552.161,Z 351.708,A -85,B 0,C 180,E1 -3141.952,E2 -3141.952} C_VEL
LIN {X 0,Y 552.235,Z 351.695,A -85,B 0,C 180,E1 -3144.889,E2 -3144.889} C_VEL
LIN {X 0,Y 552.229,Z 351.695,A -85,B 0,C 180,E1 -3147.812,E2 -3147.812} C_VEL
LIN {X 0,Y 552.246,Z 351.695,A -85,B 0,C 180,E1 -3150.729,E2 -3150.729} C_VEL
LIN {X 0,Y 552.206,Z 351.697,A -85,B 0,C 180,E1 -3152.918,E2 -3152.918} C_VEL
LIN {X 0,Y 552.205,Z 351.7,A -85,B 0,C 180,E1 -3155.844,E2 -3155.844} C_VEL
LIN {X 0,Y 552.162,Z 351.709,A -85,B 0,C 180,E1 -3158.786,E2 -3158.786} C_VEL
LIN {X 0,Y 552.167,Z 351.705,A -85,B 0,C 180,E1 -3161.751,E2 -3161.751} C_VEL
LIN {X 0,Y 552.141,Z 351.705,A -85,B 0,C 180,E1 -3164.748,E2 -3164.748} C_VEL
LIN {X 0,Y 552.113,Z 351.71,A -85,B 0,C 180,E1 -3167.789,E2 -3167.789} C_VEL
LIN {X 0,Y 552.131,Z 351.71,A -85,B 0,C 180,E1 -3170.101,E2 -3170.101} C_VEL
LIN {X 0,Y 552.097,Z 351.713,A -85,B 0,C 180,E1 -3172.451,E2 -3172.451} C_VEL
LIN {X 0,Y 552.16,Z 351.708,A -85,B 0,C 180,E1 -3175.351,E2 -3175.351} C_VEL
LIN {X 0,Y 552.124,Z 351.708,A -85,B 0,C 180,E1 -3178.098,E2 -3178.098} C_VEL
LIN {X 0,Y 552.106,Z 351.715,A -85,B 0,C 180,E1 -3180.609,E2 -3180.609} C_VEL
LIN {X 0,Y 552.127,Z 351.708,A -85,B 0,C 180,E1 -3183.185,E2 -3183.185} C_VEL
LIN {X 0,Y 552.089,Z 351.714,A -85,B 0,C 180,E1 -3185.844,E2 -3185.844} C_VEL
LIN {X 0,Y 552.121,Z 351.712,A -85,B 0,C 180,E1 -3188.589,E2 -3188.589} C_VEL
LIN {X 0,Y 552.137,Z 351.707,A -85,B 0,C 180,E1 -3191.445,E2 -3191.445} C_VEL
LIN {X 0,Y 552.098,Z 351.711,A -85,B 0,C 180,E1 -3194.532,E2 -3194.532} C_VEL
LIN {X 0,Y 552.133,Z 351.708,A -85,B 0,C 180,E1 -3197.585,E2 -3197.585} C_VEL
LIN {X 0,Y 552.137,Z 351.712,A -85,B 0,C 180,E1 -3200.473,E2 -3200.473} C_VEL
LIN {X 0,Y 552.116,Z 351.71,A -85,B 0,C 180,E1 -3203.316,E2 -3203.316} C_VEL
LIN {X 0,Y 552.133,Z 351.708,A -85,B 0,C 180,E1 -3205.939,E2 -3205.939} C_VEL
LIN {X 0,Y 552.123,Z 351.711,A -85,B 0,C 180,E1 -3208.541,E2 -3208.541} C_VEL
LIN {X 0,Y 552.168,Z 351.816,A -85,B 0,C 180,E1 -3210.164,E2 -3210.164} C_VEL
LIN {X 0,Y 552.057,Z 359.568,A -85,B 0,C 180,E1 -3213.54,E2 -3213.54} C_VEL
LIN {X 0,Y 552.005,Z 365.022,A -85,B 0,C 180,E1 -3215.957,E2 -3215.957} C_VEL
LIN {X 0,Y 551.943,Z 370.369,A -85,B 0,C 180,E1 -3218.361,E2 -3218.361} C_VEL
LIN {X 0,Y 551.867,Z 377.358,A -85,B 0,C 180,E1 -3221.435,E2 -3221.435} C_VEL
LIN {X 0,Y 551.808,Z 382.67,A -85,B 0,C 180,E1 -3223.728,E2 -3223.728} C_VEL
LIN {X 0,Y 551.776,Z 387.995,A -85,B 0,C 180,E1 -3225.995,E2 -3225.995} C_VEL
LIN {X 0,Y 551.768,Z 395.198,A -85,B 0,C 180,E1 -3228.985,E2 -3228.985} C_VEL
LIN {X 0,Y 551.729,Z 403.317,A -85,B 0,C 180,E1 -3232.314,E2 -3232.314} C_VEL
LIN {X 0,Y 551.736,Z 403.744,A -85,B 0,C 180,E1 -3232.475,E2 -3232.475} C_VEL
LIN {X 0,Y 552.173,Z 412.41,A -85,B 0,C 180,E1 -3232.789,E2 -3232.789} C_VEL
LIN {X 0,Y 552.051,Z 421.356,A -85,B 0,C 180,E1 -3233.255,E2 -3233.255} C_VEL
LIN {X 0,Y 552.007,Z 429.066,A -85,B 0,C 180,E1 -3233.787,E2 -3233.787} C_VEL
LIN {X 0,Y 551.853,Z 437.066,A -85,B 0,C 180,E1 -3234.519,E2 -3234.519} C_VEL
LIN {X 0,Y 551.905,Z 443.237,A -85,B 0,C 180,E1 -3235.252,E2 -3235.252} C_VEL
LIN {X 0,Y 551.82,Z 448.094,A -85,B 0,C 180,E1 -3235.983,E2 -3235.983} C_VEL
LIN {X 0,Y 551.785,Z 451.839,A -85,B 0,C 180,E1 -3236.714,E2 -3236.714} C_VEL
LIN {X 0,Y 551.675,Z 455.843,A -85,B 0,C 180,E1 -3237.81,E2 -3237.81} C_VEL
LIN {X 0,Y 551.649,Z 457.582,A -85,B 0,C 180,E1 -3238.54,E2 -3238.54} C_VEL
LIN {X 0,Y 551.642,Z 458.623,A -85,B 0,C 180,E1 -3239.27,E2 -3239.27} C_VEL
LIN {X 0,Y 551.641,Z 458.996,A -85,B 0,C 180,E1 -3240,E2 -3240} C_VEL
LIN {X 0,Y 551.642,Z 458.71,A -85,B 0,C 180,E1 -3240.73,E2 -3240.73} C_VEL
LIN {X 0,Y 551.648,Z 457.759,A -85,B 0,C 180,E1 -3241.46,E2 -3241.46} C_VEL
LIN {X 0,Y 551.674,Z 456.117,A -85,B 0,C 180,E1 -3242.19,E2 -3242.19} C_VEL
LIN {X 0,Y 551.742,Z 453.728,A -85,B 0,C 180,E1 -3242.921,E2 -3242.921} C_VEL
LIN {X 0,Y 551.8,Z 448.595,A -85,B 0,C 180,E1 -3244.017,E2 -3244.017} C_VEL
LIN {X 0,Y 551.887,Z 442.518,A -85,B 0,C 180,E1 -3244.931,E2 -3244.931} C_VEL
LIN {X 0,Y 551.869,Z 436.2,A -85,B 0,C 180,E1 -3245.664,E2 -3245.664} C_VEL
LIN {X 0,Y 552.006,Z 429.045,A -85,B 0,C 180,E1 -3246.304,E2 -3246.304} C_VEL
LIN {X 0,Y 552.035,Z 421.178,A -85,B 0,C 180,E1 -3246.846,E2 -3246.846} C_VEL
LIN {X 0,Y 552.154,Z 412.152,A -85,B 0,C 180,E1 -3247.313,E2 -3247.313} C_VEL
LIN {X 0,Y 551.719,Z 403.651,A -85,B 0,C 180,E1 -3247.64,E2 -3247.64} C_VEL
LIN {X 0,Y 551.767,Z 395.417,A -85,B 0,C 180,E1 -3251.015,E2 -3251.015} C_VEL
LIN {X 0,Y 551.767,Z 388.248,A -85,B 0,C 180,E1 -3254.005,E2 -3254.005} C_VEL
LIN {X 0,Y 551.875,Z 381.388,A -85,B 0,C 180,E1 -3257.032,E2 -3257.032} C_VEL
LIN {X 0,Y 551.955,Z 375.78,A -85,B 0,C 180,E1 -3259.569,E2 -3259.569} C_VEL
LIN {X 0,Y 552.047,Z 371.241,A -85,B 0,C 180,E1 -3261.666,E2 -3261.666} C_VEL
LIN {X 0,Y 552.034,Z 365.591,A -85,B 0,C 180,E1 -3264.041,E2 -3264.041} C_VEL
LIN {X 0,Y 552.129,Z 360.133,A -85,B 0,C 180,E1 -3266.456,E2 -3266.456} C_VEL
LIN {X 0,Y 552.222,Z 352.559,A -85,B 0,C 180,E1 -3269.759,E2 -3269.759} C_VEL
LIN {X 0,Y 552.245,Z 351.699,A -85,B 0,C 180,E1 -3270.146,E2 -3270.146} C_VEL
LIN {X 0,Y 552.119,Z 351.713,A -85,B 0,C 180,E1 -3273.186,E2 -3273.186} C_VEL
LIN {X 0,Y 552.09,Z 351.719,A -85,B 0,C 180,E1 -3275.844,E2 -3275.844} C_VEL
LIN {X 0,Y 552.13,Z 351.714,A -85,B 0,C 180,E1 -3279.062,E2 -3279.062} C_VEL
LIN {X 0,Y 552.144,Z 351.71,A -85,B 0,C 180,E1 -3281.444,E2 -3281.444} C_VEL
LIN {X 0,Y 552.101,Z 351.716,A -85,B 0,C 180,E1 -3284.532,E2 -3284.532} C_VEL
LIN {X 0,Y 552.135,Z 351.712,A -85,B 0,C 180,E1 -3287.584,E2 -3287.584} C_VEL
LIN {X 0,Y 552.132,Z 351.713,A -85,B 0,C 180,E1 -3290.473,E2 -3290.473} C_VEL
LIN {X 0,Y 552.11,Z 351.714,A -85,B 0,C 180,E1 -3293.317,E2 -3293.317} C_VEL
LIN {X 0,Y 552.131,Z 351.714,A -85,B 0,C 180,E1 -3295.939,E2 -3295.939} C_VEL
LIN {X 0,Y 552.123,Z 351.715,A -85,B 0,C 180,E1 -3298.541,E2 -3298.541} C_VEL
LIN {X 0,Y 552.189,Z 351.871,A -85,B 0,C 180,E1 -3300.344,E2 -3300.344} C_VEL
LIN {X 0,Y 553.827,Z 359.694,A -85,B 0,C 180,E1 -3301.996,E2 -3301.996} C_VEL
LIN {X 0,Y 553.469,Z 370.812,A -85,B 0,C 180,E1 -3304.059,E2 -3304.059} C_VEL
LIN {X 0,Y 553.088,Z 384.511,A -85,B 0,C 180,E1 -3306.489,E2 -3306.489} C_VEL
LIN {X 0,Y 552.857,Z 400.527,A -85,B 0,C 180,E1 -3309.149,E2 -3309.149} C_VEL
LIN {X 0,Y 552.574,Z 419.132,A -85,B 0,C 180,E1 -3312.227,E2 -3312.227} C_VEL
LIN {X 0,Y 552.324,Z 436.557,A -85,B 0,C 180,E1 -3315.087,E2 -3315.087} C_VEL
LIN {X 0,Y 552.208,Z 447.98,A -85,B 0,C 180,E1 -3316.944,E2 -3316.944} C_VEL
LIN {X 0,Y 553.128,Z 454.937,A -85,B 0,C 180,E1 -3317.082,E2 -3317.082} C_VEL
LIN {X 0,Y 553.023,Z 468.212,A -85,B 0,C 180,E1 -3317.407,E2 -3317.407} C_VEL
LIN {X 0,Y 552.838,Z 479.915,A -85,B 0,C 180,E1 -3317.826,E2 -3317.826} C_VEL
LIN {X 0,Y 552.712,Z 490.92,A -85,B 0,C 180,E1 -3318.354,E2 -3318.354} C_VEL
LIN {X 0,Y 552.544,Z 501.585,A -85,B 0,C 180,E1 -3319.001,E2 -3319.001} C_VEL
LIN {X 0,Y 552.311,Z 512.468,A -85,B 0,C 180,E1 -3319.831,E2 -3319.831} C_VEL
LIN {X 0,Y 552.131,Z 523.111,A -85,B 0,C 180,E1 -3320.845,E2 -3320.845} C_VEL
LIN {X 0,Y 552.013,Z 530.959,A -85,B 0,C 180,E1 -3321.765,E2 -3321.765} C_VEL
LIN {X 0,Y 551.889,Z 538.62,A -85,B 0,C 180,E1 -3322.868,E2 -3322.868} C_VEL
LIN {X 0,Y 551.867,Z 545.679,A -85,B 0,C 180,E1 -3324.152,E2 -3324.152} C_VEL
LIN {X 0,Y 551.725,Z 550.372,A -85,B 0,C 180,E1 -3325.25,E2 -3325.25} C_VEL
LIN {X 0,Y 551.75,Z 553.957,A -85,B 0,C 180,E1 -3326.348,E2 -3326.348} C_VEL
LIN {X 0,Y 551.723,Z 555.807,A -85,B 0,C 180,E1 -3327.079,E2 -3327.079} C_VEL
LIN {X 0,Y 551.645,Z 558.184,A -85,B 0,C 180,E1 -3328.54,E2 -3328.54} C_VEL
LIN {X 0,Y 551.64,Z 559,A -85,B 0,C 180,E1 -3330,E2 -3330} C_VEL
LIN {X 0,Y 551.645,Z 558.185,A -85,B 0,C 180,E1 -3331.46,E2 -3331.46} C_VEL
LIN {X 0,Y 551.723,Z 555.81,A -85,B 0,C 180,E1 -3332.921,E2 -3332.921} C_VEL
LIN {X 0,Y 551.763,Z 552.897,A -85,B 0,C 180,E1 -3334.017,E2 -3334.017} C_VEL
LIN {X 0,Y 551.724,Z 548.95,A -85,B 0,C 180,E1 -3335.116,E2 -3335.116} C_VEL
LIN {X 0,Y 551.814,Z 543.128,A -85,B 0,C 180,E1 -3336.352,E2 -3336.352} C_VEL
LIN {X 0,Y 551.926,Z 536.238,A -85,B 0,C 180,E1 -3337.499,E2 -3337.499} C_VEL
LIN {X 0,Y 552.082,Z 527.993,A -85,B 0,C 180,E1 -3338.602,E2 -3338.602} C_VEL
LIN {X 0,Y 552.201,Z 519.54,A -85,B 0,C 180,E1 -3339.524,E2 -3339.524} C_VEL
LIN {X 0,Y 552.426,Z 509.095,A -85,B 0,C 180,E1 -3340.445,E2 -3340.445} C_VEL
LIN {X 0,Y 552.594,Z 498.132,A -85,B 0,C 180,E1 -3341.224,E2 -3341.224} C_VEL
LIN {X 0,Y 552.751,Z 487.41,A -85,B 0,C 180,E1 -3341.831,E2 -3341.831} C_VEL
LIN {X 0,Y 552.899,Z 475.766,A -85,B 0,C 180,E1 -3342.34,E2 -3342.34} C_VEL
LIN {X 0,Y 553.048,Z 462.349,A -85,B 0,C 180,E1 -3342.756,E2 -3342.756} C_VEL
LIN {X 0,Y 552.939,Z 453.071,A -85,B 0,C 180,E1 -3342.954,E2 -3342.954} C_VEL
LIN {X 0,Y 552.208,Z 447.982,A -85,B 0,C 180,E1 -3343.056,E2 -3343.056} C_VEL
LIN {X 0,Y 552.432,Z 429.519,A -85,B 0,C 180,E1 -3346.063,E2 -3346.063} C_VEL
LIN {X 0,Y 552.687,Z 411.056,A -85,B 0,C 180,E1 -3349.113,E2 -3349.113} C_VEL
LIN {X 0,Y 552.91,Z 397.148,A -85,B 0,C 180,E1 -3351.435,E2 -3351.435} C_VEL
LIN {X 0,Y 553.234,Z 382.257,A -85,B 0,C 180,E1 -3353.986,E2 -3353.986} C_VEL
LIN {X 0,Y 553.672,Z 365.055,A -85,B 0,C 180,E1 -3356.987,E2 -3356.987} C_VEL
LIN {X 0,Y 553.704,Z 359.313,A -85,B 0,C 180,E1 -3358.01,E2 -3358.01} C_VEL
LIN {X 0,Y 552.121,Z 351.713,A -85,B 0,C 180,E1 -3359.502,E2 -3359.502} C_VEL
LIN {X 0,Y 552.129,Z 351.71,A -85,B 0,C 180,E1 -3362.318,E2 -3362.318} C_VEL
LIN {X 0,Y 552.087,Z 351.717,A -85,B 0,C 180,E1 -3364.949,E2 -3364.949} C_VEL
LIN {X 0,Y 552.098,Z 351.711,A -85,B 0,C 180,E1 -3367.886,E2 -3367.886} C_VEL
LIN {X 0,Y 552.112,Z 351.712,A -85,B 0,C 180,E1 -3370.481,E2 -3370.481} C_VEL
LIN {X 0,Y 552.117,Z 351.714,A -85,B 0,C 180,E1 -3373.484,E2 -3373.484} C_VEL
LIN {X 0,Y 552.122,Z 351.712,A -85,B 0,C 180,E1 -3376.578,E2 -3376.578} C_VEL
LIN {X 0,Y 552.121,Z 351.708,A -85,B 0,C 180,E1 -3379.52,E2 -3379.52} C_VEL
LIN {X 0,Y 552.096,Z 351.712,A -85,B 0,C 180,E1 -3382.336,E2 -3382.336} C_VEL
LIN {X 0,Y 552.123,Z 351.713,A -85,B 0,C 180,E1 -3385.054,E2 -3385.054} C_VEL
LIN {X 0,Y 552.119,Z 351.709,A -85,B 0,C 180,E1 -3387.681,E2 -3387.681} C_VEL
LIN {X 0,Y 552.115,Z 351.715,A -85,B 0,C 180,E1 -3390.235,E2 -3390.235} C_VEL
LIN {X 0,Y 552.142,Z 351.706,A -85,B 0,C 180,E1 -3393,E2 -3393} C_VEL
LIN {X 0,Y 552.115,Z 351.714,A -85,B 0,C 180,E1 -3395.161,E2 -3395.161} C_VEL
LIN {X 0,Y 552.127,Z 351.712,A -85,B 0,C 180,E1 -3398.337,E2 -3398.337} C_VEL
LIN {X 0,Y 552.157,Z 351.705,A -85,B 0,C 180,E1 -3400.674,E2 -3400.674} C_VEL
LIN {X 0,Y 552.119,Z 351.713,A -85,B 0,C 180,E1 -3403.737,E2 -3403.737} C_VEL
LIN {X 0,Y 552.139,Z 351.706,A -85,B 0,C 180,E1 -3406.005,E2 -3406.005} C_VEL
LIN {X 0,Y 552.165,Z 351.705,A -85,B 0,C 180,E1 -3408.993,E2 -3408.993} C_VEL
LIN {X 0,Y 552.16,Z 351.709,A -85,B 0,C 180,E1 -3411.952,E2 -3411.952} C_VEL
LIN {X 0,Y 552.232,Z 351.696,A -85,B 0,C 180,E1 -3414.889,E2 -3414.889} C_VEL
LIN {X 0,Y 552.222,Z 351.696,A -85,B 0,C 180,E1 -3417.812,E2 -3417.812} C_VEL
LIN {X 0,Y 552.245,Z 351.694,A -85,B 0,C 180,E1 -3420.729,E2 -3420.729} C_VEL
LIN {X 0,Y 552.207,Z 351.697,A -85,B 0,C 180,E1 -3422.918,E2 -3422.918} C_VEL
LIN {X 0,Y 552.2,Z 351.699,A -85,B 0,C 180,E1 -3425.844,E2 -3425.844} C_VEL
LIN {X 0,Y 552.165,Z 351.707,A -85,B 0,C 180,E1 -3428.786,E2 -3428.786} C_VEL
LIN {X 0,Y 552.165,Z 351.707,A -85,B 0,C 180,E1 -3431.75,E2 -3431.75} C_VEL
LIN {X 0,Y 552.138,Z 351.707,A -85,B 0,C 180,E1 -3434.748,E2 -3434.748} C_VEL
LIN {X 0,Y 552.113,Z 351.709,A -85,B 0,C 180,E1 -3437.788,E2 -3437.788} C_VEL
LIN {X 0,Y 552.133,Z 351.711,A -85,B 0,C 180,E1 -3440.101,E2 -3440.101} C_VEL
LIN {X 0,Y 552.097,Z 351.712,A -85,B 0,C 180,E1 -3442.451,E2 -3442.451} C_VEL
LIN {X 0,Y 552.157,Z 351.709,A -85,B 0,C 180,E1 -3445.35,E2 -3445.35} C_VEL
LIN {X 0,Y 552.111,Z 351.71,A -85,B 0,C 180,E1 -3448.098,E2 -3448.098} C_VEL
LIN {X 0,Y 552.104,Z 351.713,A -85,B 0,C 180,E1 -3450.613,E2 -3450.613} C_VEL
LIN {X 0,Y 552.125,Z 351.71,A -85,B 0,C 180,E1 -3453.185,E2 -3453.185} C_VEL
LIN {X 0,Y 552.116,Z 351.709,A -85,B 0,C 180,E1 -3453.793,E2 -3453.793} C_VEL
LIN {X 0,Y 551.48,Z 351.792,A -85,B 0,C 180,E1 -3454.401,E2 -3454.401} C_VEL
LIN {X 0,Y 548.657,Z 352.15,A -85,B 0,C 180,E1 -3455.389,E2 -3455.389} C_VEL
LIN {X 0,Y 546.236,Z 352.452,A -85,B 0,C 180,E1 -3456.185,E2 -3456.185} C_VEL
LIN {X 0,Y 545.167,Z 352.582,A -85,B 0,C 180,E1 -3456.799,E2 -3456.799} C_VEL
LIN {X 0,Y 545.065,Z 352.592,A -85,B 0,C 180,E1 -3457.007,E2 -3457.007} C_VEL
LIN {X 0,Y 545.074,Z 352.59,A -85,B 0,C 180,E1 -3460.142,E2 -3460.142} C_VEL
LIN {X 0,Y 545.065,Z 352.588,A -85,B 0,C 180,E1 -3462.697,E2 -3462.697} C_VEL
LIN {X 0,Y 545.065,Z 352.592,A -85,B 0,C 180,E1 -3465.167,E2 -3465.167} C_VEL
LIN {X 0,Y 545.084,Z 352.584,A -85,B 0,C 180,E1 -3467.898,E2 -3467.898} C_VEL
LIN {X 0,Y 545.082,Z 352.586,A -85,B 0,C 180,E1 -3470.819,E2 -3470.819} C_VEL
LIN {X 0,Y 545.044,Z 352.595,A -85,B 0,C 180,E1 -3473.62,E2 -3473.62} C_VEL
LIN {X 0,Y 545.071,Z 352.587,A -85,B 0,C 180,E1 -3476.329,E2 -3476.329} C_VEL
LIN {X 0,Y 545.068,Z 352.589,A -85,B 0,C 180,E1 -3478.952,E2 -3478.952} C_VEL
LIN {X 0,Y 545.107,Z 352.583,A -85,B 0,C 180,E1 -3481.508,E2 -3481.508} C_VEL
LIN {X 0,Y 545.098,Z 352.583,A -85,B 0,C 180,E1 -3484.491,E2 -3484.491} C_VEL
LIN {X 0,Y 545.042,Z 352.594,A -85,B 0,C 180,E1 -3487.243,E2 -3487.243} C_VEL
LIN {X 0,Y 545.124,Z 352.586,A -85,B 0,C 180,E1 -3490.415,E2 -3490.415} C_VEL
LIN {X 0,Y 545.078,Z 352.59,A -85,B 0,C 180,E1 -3493.521,E2 -3493.521} C_VEL
LIN {X 0,Y 545.099,Z 352.585,A -85,B 0,C 180,E1 -3495.82,E2 -3495.82} C_VEL
LIN {X 0,Y 545.122,Z 352.584,A -85,B 0,C 180,E1 -3498.85,E2 -3498.85} C_VEL
LIN {X 0,Y 545.132,Z 352.582,A -85,B 0,C 180,E1 -3501.847,E2 -3501.847} C_VEL
LIN {X 0,Y 545.21,Z 352.57,A -85,B 0,C 180,E1 -3504.823,E2 -3504.823} C_VEL
LIN {X 0,Y 545.2,Z 352.571,A -85,B 0,C 180,E1 -3507.784,E2 -3507.784} C_VEL
LIN {X 0,Y 545.216,Z 352.57,A -85,B 0,C 180,E1 -3510.739,E2 -3510.739} C_VEL
LIN {X 0,Y 545.173,Z 352.573,A -85,B 0,C 180,E1 -3512.956,E2 -3512.956} C_VEL
LIN {X 0,Y 545.176,Z 352.575,A -85,B 0,C 180,E1 -3515.92,E2 -3515.92} C_VEL
LIN {X 0,Y 545.121,Z 352.585,A -85,B 0,C 180,E1 -3518.9,E2 -3518.9} C_VEL
LIN {X 0,Y 545.139,Z 352.582,A -85,B 0,C 180,E1 -3521.904,E2 -3521.904} C_VEL
LIN {X 0,Y 545.09,Z 352.585,A -85,B 0,C 180,E1 -3524.944,E2 -3524.944} C_VEL
LIN {X 0,Y 545.081,Z 352.586,A -85,B 0,C 180,E1 -3528.026,E2 -3528.026} C_VEL
LIN {X 0,Y 545.097,Z 352.589,A -85,B 0,C 180,E1 -3530.372,E2 -3530.372} C_VEL
LIN {X 0,Y 545.085,Z 352.588,A -85,B 0,C 180,E1 -3533.559,E2 -3533.559} C_VEL
LIN {X 0,Y 545.084,Z 352.585,A -85,B 0,C 180,E1 -3536.001,E2 -3536.001} C_VEL
LIN {X 0,Y 545.094,Z 352.589,A -85,B 0,C 180,E1 -3538.748,E2 -3538.748} C_VEL
LIN {X 0,Y 545.063,Z 352.589,A -85,B 0,C 180,E1 -3541.679,E2 -3541.679} C_VEL
LIN {X 0,Y 545.079,Z 352.586,A -85,B 0,C 180,E1 -3544.392,E2 -3544.392} C_VEL
LIN {X 0,Y 545.04,Z 352.595,A -85,B 0,C 180,E1 -3547.304,E2 -3547.304} C_VEL
LIN {X 0,Y 545.07,Z 352.59,A -85,B 0,C 180,E1 -3550.143,E2 -3550.143} C_VEL
LIN {X 0,Y 545.091,Z 352.584,A -85,B 0,C 180,E1 -3553.106,E2 -3553.106} C_VEL
LIN {X 0,Y 545.053,Z 352.588,A -85,B 0,C 180,E1 -3556.226,E2 -3556.226} C_VEL
LIN {X 0,Y 545.085,Z 352.591,A -85,B 0,C 180,E1 -3558.885,E2 -3558.885} C_VEL
LIN {X 0,Y 545.088,Z 352.587,A -85,B 0,C 180,E1 -3560.819,E2 -3560.819} C_VEL
LIN {X 0,Y 545.055,Z 352.593,A -85,B 0,C 180,E1 -3563.62,E2 -3563.62} C_VEL
LIN {X 0,Y 545.071,Z 352.586,A -85,B 0,C 180,E1 -3566.328,E2 -3566.328} C_VEL
LIN {X 0,Y 545.084,Z 352.591,A -85,B 0,C 180,E1 -3568.953,E2 -3568.953} C_VEL
LIN {X 0,Y 545.131,Z 352.69,A -85,B 0,C 180,E1 -3570.134,E2 -3570.134} C_VEL
LIN {X 0,Y 545.029,Z 359.576,A -85,B 0,C 180,E1 -3573.172,E2 -3573.172} C_VEL
LIN {X 0,Y 544.968,Z 365.141,A -85,B 0,C 180,E1 -3575.627,E2 -3575.627} C_VEL
LIN {X 0,Y 544.892,Z 370.84,A -85,B 0,C 180,E1 -3578.227,E2 -3578.227} C_VEL
LIN {X 0,Y 544.794,Z 377.473,A -85,B 0,C 180,E1 -3581.185,E2 -3581.185} C_VEL
LIN {X 0,Y 544.758,Z 382.783,A -85,B 0,C 180,E1 -3583.511,E2 -3583.511} C_VEL
LIN {X 0,Y 544.701,Z 388.108,A -85,B 0,C 180,E1 -3585.809,E2 -3585.809} C_VEL
LIN {X 0,Y 544.686,Z 395.228,A -85,B 0,C 180,E1 -3588.84,E2 -3588.84} C_VEL
LIN {X 0,Y 544.654,Z 403.544,A -85,B 0,C 180,E1 -3592.306,E2 -3592.306} C_VEL
LIN {X 0,Y 544.632,Z 403.765,A -85,B 0,C 180,E1 -3592.376,E2 -3592.376} C_VEL
LIN {X 0,Y 545.14,Z 412.423,A -85,B 0,C 180,E1 -3592.695,E2 -3592.695} C_VEL
LIN {X 0,Y 545.02,Z 420.185,A -85,B 0,C 180,E1 -3593.095,E2 -3593.095} C_VEL
LIN {X 0,Y 544.971,Z 427.63,A -85,B 0,C 180,E1 -3593.597,E2 -3593.597} C_VEL
LIN {X 0,Y 544.818,Z 435.336,A -85,B 0,C 180,E1 -3594.262,E2 -3594.262} C_VEL
LIN {X 0,Y 544.812,Z 441.825,A -85,B 0,C 180,E1 -3595.005,E2 -3595.005} C_VEL
LIN {X 0,Y 544.739,Z 446.952,A -85,B 0,C 180,E1 -3595.746,E2 -3595.746} C_VEL
LIN {X 0,Y 544.713,Z 451.842,A -85,B 0,C 180,E1 -3596.672,E2 -3596.672} C_VEL
LIN {X 0,Y 544.59,Z 455.845,A -85,B 0,C 180,E1 -3597.781,E2 -3597.781} C_VEL
LIN {X 0,Y 544.55,Z 457.584,A -85,B 0,C 180,E1 -3598.521,E2 -3598.521} C_VEL
LIN {X 0,Y 544.543,Z 458.624,A -85,B 0,C 180,E1 -3599.26,E2 -3599.26} C_VEL
LIN {X 0,Y 544.541,Z 458.996,A -85,B 0,C 180,E1 -3600,E2 -3600} C_VEL
LIN {X 0,Y 544.542,Z 458.709,A -85,B 0,C 180,E1 -3600.739,E2 -3600.739} C_VEL
LIN {X 0,Y 544.549,Z 457.757,A -85,B 0,C 180,E1 -3601.479,E2 -3601.479} C_VEL
LIN {X 0,Y 544.589,Z 456.115,A -85,B 0,C 180,E1 -3602.219,E2 -3602.219} C_VEL
LIN {X 0,Y 544.672,Z 453.726,A -85,B 0,C 180,E1 -3602.959,E2 -3602.959} C_VEL
LIN {X 0,Y 544.721,Z 448.593,A -85,B 0,C 180,E1 -3604.069,E2 -3604.069} C_VEL
LIN {X 0,Y 544.796,Z 442.513,A -85,B 0,C 180,E1 -3604.995,E2 -3604.995} C_VEL
LIN {X 0,Y 544.817,Z 436.194,A -85,B 0,C 180,E1 -3605.738,E2 -3605.738} C_VEL
LIN {X 0,Y 544.964,Z 428.761,A -85,B 0,C 180,E1 -3606.407,E2 -3606.407} C_VEL
LIN {X 0,Y 545,Z 420.532,A -85,B 0,C 180,E1 -3606.974,E2 -3606.974} C_VEL
LIN {X 0,Y 545.151,Z 410.966,A -85,B 0,C 180,E1 -3607.454,E2 -3607.454} C_VEL
LIN {X 0,Y 544.635,Z 403.649,A -85,B 0,C 180,E1 -3607.74,E2 -3607.74} C_VEL
LIN {X 0,Y 544.686,Z 395.512,A -85,B 0,C 180,E1 -3611.16,E2 -3611.16} C_VEL
LIN {X 0,Y 544.71,Z 388.588,A -85,B 0,C 180,E1 -3614.19,E2 -3614.19} C_VEL
LIN {X 0,Y 544.852,Z 381.54,A -85,B 0,C 180,E1 -3617.345,E2 -3617.345} C_VEL
LIN {X 0,Y 544.921,Z 374.957,A -85,B 0,C 180,E1 -3620.379,E2 -3620.379} C_VEL
LIN {X 0,Y 544.971,Z 369.409,A -85,B 0,C 180,E1 -3622.761,E2 -3622.761} C_VEL
LIN {X 0,Y 545.078,Z 362.209,A -85,B 0,C 180,E1 -3626.001,E2 -3626.001} C_VEL
LIN {X 0,Y 545.141,Z 355.966,A -85,B 0,C 180,E1 -3628.757,E2 -3628.757} C_VEL
LIN {X 0,Y 545.196,Z 352.578,A -85,B 0,C 180,E1 -3630.267,E2 -3630.267} C_VEL
LIN {X 0,Y 545.07,Z 352.593,A -85,B 0,C 180,E1 -3633.672,E2 -3633.672} C_VEL
LIN {X 0,Y 545.074,Z 352.592,A -85,B 0,C 180,E1 -3636.926,E2 -3636.926} C_VEL
LIN {X 0,Y 545.097,Z 352.589,A -85,B 0,C 180,E1 -3640.14,E2 -3640.14} C_VEL
LIN {X 0,Y 545.091,Z 352.59,A -85,B 0,C 180,E1 -3643.106,E2 -3643.106} C_VEL
LIN {X 0,Y 545.069,Z 352.592,A -85,B 0,C 180,E1 -3646.224,E2 -3646.224} C_VEL
LIN {X 0,Y 545.091,Z 352.589,A -85,B 0,C 180,E1 -3648.886,E2 -3648.886} C_VEL
LIN {X 0,Y 545.054,Z 352.595,A -85,B 0,C 180,E1 -3651.762,E2 -3651.762} C_VEL
LIN {X 0,Y 545.04,Z 352.596,A -85,B 0,C 180,E1 -3654.532,E2 -3654.532} C_VEL
LIN {X 0,Y 545.085,Z 352.592,A -85,B 0,C 180,E1 -3657.212,E2 -3657.212} C_VEL
LIN {X 0,Y 545.124,Z 352.783,A -85,B 0,C 180,E1 -3660.027,E2 -3660.027} C_VEL
LIN {X 0,Y 546.899,Z 360.922,A -85,B 0,C 180,E1 -3661.819,E2 -3661.819} C_VEL
LIN {X 0,Y 546.697,Z 370.605,A -85,B 0,C 180,E1 -3663.672,E2 -3663.672} C_VEL
LIN {X 0,Y 546.116,Z 388.455,A -85,B 0,C 180,E1 -3666.889,E2 -3666.889} C_VEL
LIN {X 0,Y 545.794,Z 406.495,A -85,B 0,C 180,E1 -3669.911,E2 -3669.911} C_VEL
LIN {X 0,Y 545.511,Z 424.902,A -85,B 0,C 180,E1 -3672.956,E2 -3672.956} C_VEL
LIN {X 0,Y 545.248,Z 443.364,A -85,B 0,C 180,E1 -3676.014,E2 -3676.014} C_VEL
LIN {X 0,Y 545.196,Z 448.077,A -85,B 0,C 180,E1 -3676.783,E2 -3676.783} C_VEL
LIN {X 0,Y 546.177,Z 456.078,A -85,B 0,C 180,E1 -3676.939,E2 -3676.939} C_VEL
LIN {X 0,Y 546.035,Z 469.736,A -85,B 0,C 180,E1 -3677.29,E2 -3677.29} C_VEL
LIN {X 0,Y 545.877,Z 482.507,A -85,B 0,C 180,E1 -3677.782,E2 -3677.782} C_VEL
LIN {X 0,Y 545.686,Z 493.535,A -85,B 0,C 180,E1 -3678.351,E2 -3678.351} C_VEL
LIN {X 0,Y 545.494,Z 505.484,A -85,B 0,C 180,E1 -3679.139,E2 -3679.139} C_VEL
LIN {X 0,Y 545.282,Z 515.644,A -85,B 0,C 180,E1 -3679.979,E2 -3679.979} C_VEL
LIN {X 0,Y 545.082,Z 524.784,A -85,B 0,C 180,E1 -3680.912,E2 -3680.912} C_VEL
LIN {X 0,Y 544.917,Z 533.687,A -85,B 0,C 180,E1 -3682.03,E2 -3682.03} C_VEL
LIN {X 0,Y 544.785,Z 540.848,A -85,B 0,C 180,E1 -3683.146,E2 -3683.146} C_VEL
LIN {X 0,Y 544.741,Z 547.365,A -85,B 0,C 180,E1 -3684.447,E2 -3684.447} C_VEL
LIN {X 0,Y 544.66,Z 551.676,A -85,B 0,C 180,E1 -3685.56,E2 -3685.56} C_VEL
LIN {X 0,Y 544.669,Z 553.958,A -85,B 0,C 180,E1 -3686.301,E2 -3686.301} C_VEL
LIN {X 0,Y 544.65,Z 555.807,A -85,B 0,C 180,E1 -3687.041,E2 -3687.041} C_VEL
LIN {X 0,Y 544.546,Z 558.183,A -85,B 0,C 180,E1 -3688.521,E2 -3688.521} C_VEL
LIN {X 0,Y 544.541,Z 559,A -85,B 0,C 180,E1 -3690,E2 -3690} C_VEL
LIN {X 0,Y 544.546,Z 558.185,A -85,B 0,C 180,E1 -3691.479,E2 -3691.479} C_VEL
LIN {X 0,Y 544.65,Z 555.81,A -85,B 0,C 180,E1 -3692.958,E2 -3692.958} C_VEL
LIN {X 0,Y 544.683,Z 552.897,A -85,B 0,C 180,E1 -3694.069,E2 -3694.069} C_VEL
LIN {X 0,Y 544.653,Z 548.95,A -85,B 0,C 180,E1 -3695.182,E2 -3695.182} C_VEL
LIN {X 0,Y 544.729,Z 543.648,A -85,B 0,C 180,E1 -3696.339,E2 -3696.339} C_VEL
LIN {X 0,Y 544.836,Z 537.466,A -85,B 0,C 180,E1 -3697.411,E2 -3697.411} C_VEL
LIN {X 0,Y 545.006,Z 529.479,A -85,B 0,C 180,E1 -3698.528,E2 -3698.528} C_VEL
LIN {X 0,Y 545.142,Z 521.335,A -85,B 0,C 180,E1 -3699.461,E2 -3699.461} C_VEL
LIN {X 0,Y 545.373,Z 511.401,A -85,B 0,C 180,E1 -3700.394,E2 -3700.394} C_VEL
LIN {X 0,Y 545.561,Z 500.539,A -85,B 0,C 180,E1 -3701.211,E2 -3701.211} C_VEL
LIN {X 0,Y 545.763,Z 489.174,A -85,B 0,C 180,E1 -3701.89,E2 -3701.89} C_VEL
LIN {X 0,Y 545.951,Z 476.977,A -85,B 0,C 180,E1 -3702.452,E2 -3702.452} C_VEL
LIN {X 0,Y 546.117,Z 464.177,A -85,B 0,C 180,E1 -3702.873,E2 -3702.873} C_VEL
LIN {X 0,Y 545.979,Z 453.614,A -85,B 0,C 180,E1 -3703.113,E2 -3703.113} C_VEL
LIN {X 0,Y 545.177,Z 447.982,A -85,B 0,C 180,E1 -3703.227,E2 -3703.227} C_VEL
LIN {X 0,Y 545.405,Z 430.673,A -85,B 0,C 180,E1 -3706.084,E2 -3706.084} C_VEL
LIN {X 0,Y 545.671,Z 413.173,A -85,B 0,C 180,E1 -3708.978,E2 -3708.978} C_VEL
LIN {X 0,Y 545.927,Z 399.203,A -85,B 0,C 180,E1 -3711.326,E2 -3711.326} C_VEL
LIN {X 0,Y 546.284,Z 383.816,A -85,B 0,C 180,E1 -3714.017,E2 -3714.017} C_VEL
LIN {X 0,Y 546.745,Z 367.24,A -85,B 0,C 180,E1 -3716.943,E2 -3716.943} C_VEL
LIN {X 0,Y 546.737,Z 360.349,A -85,B 0,C 180,E1 -3718.19,E2 -3718.19} C_VEL
LIN {X 0,Y 545.095,Z 352.589,A -85,B 0,C 180,E1 -3719.761,E2 -3719.761} C_VEL
LIN {X 0,Y 545.092,Z 352.587,A -85,B 0,C 180,E1 -3723.064,E2 -3723.064} C_VEL
LIN {X 0,Y 545.036,Z 352.592,A -85,B 0,C 180,E1 -3725.673,E2 -3725.673} C_VEL
LIN {X 0,Y 545.054,Z 352.592,A -85,B 0,C 180,E1 -3728.237,E2 -3728.237} C_VEL
LIN {X 0,Y 545.09,Z 352.584,A -85,B 0,C 180,E1 -3731.114,E2 -3731.114} C_VEL
LIN {X 0,Y 545.061,Z 352.589,A -85,B 0,C 180,E1 -3734.129,E2 -3734.129} C_VEL
LIN {X 0,Y 545.088,Z 352.589,A -85,B 0,C 180,E1 -3736.894,E2 -3736.894} C_VEL
LIN {X 0,Y 545.073,Z 352.588,A -85,B 0,C 180,E1 -3739.858,E2 -3739.858} C_VEL
LIN {X 0,Y 545.08,Z 352.587,A -85,B 0,C 180,E1 -3743.073,E2 -3743.073} C_VEL
LIN {X 0,Y 545.069,Z 352.588,A -85,B 0,C 180,E1 -3746.328,E2 -3746.328} C_VEL
LIN {X 0,Y 545.07,Z 352.588,A -85,B 0,C 180,E1 -3748.952,E2 -3748.952} C_VEL
LIN {X 0,Y 545.105,Z 352.584,A -85,B 0,C 180,E1 -3751.508,E2 -3751.508} C_VEL
LIN {X 0,Y 545.097,Z 352.583,A -85,B 0,C 180,E1 -3754.491,E2 -3754.491} C_VEL
LIN {X 0,Y 545.038,Z 352.593,A -85,B 0,C 180,E1 -3757.242,E2 -3757.242} C_VEL
LIN {X 0,Y 545.122,Z 352.584,A -85,B 0,C 180,E1 -3760.415,E2 -3760.415} C_VEL
LIN {X 0,Y 545.076,Z 352.591,A -85,B 0,C 180,E1 -3763.521,E2 -3763.521} C_VEL
LIN {X 0,Y 545.098,Z 352.584,A -85,B 0,C 180,E1 -3765.82,E2 -3765.82} C_VEL
LIN {X 0,Y 545.12,Z 352.584,A -85,B 0,C 180,E1 -3768.849,E2 -3768.849} C_VEL
LIN {X 0,Y 545.13,Z 352.585,A -85,B 0,C 180,E1 -3771.847,E2 -3771.847} C_VEL
LIN {X 0,Y 545.207,Z 352.571,A -85,B 0,C 180,E1 -3774.823,E2 -3774.823} C_VEL
LIN {X 0,Y 545.195,Z 352.571,A -85,B 0,C 180,E1 -3777.784,E2 -3777.784} C_VEL
LIN {X 0,Y 545.215,Z 352.57,A -85,B 0,C 180,E1 -3780.739,E2 -3780.739} C_VEL
LIN {X 0,Y 545.174,Z 352.574,A -85,B 0,C 180,E1 -3782.956,E2 -3782.956} C_VEL
LIN {X 0,Y 545.172,Z 352.574,A -85,B 0,C 180,E1 -3785.92,E2 -3785.92} C_VEL
LIN {X 0,Y 545.123,Z 352.583,A -85,B 0,C 180,E1 -3788.9,E2 -3788.9} C_VEL
LIN {X 0,Y 545.137,Z 352.584,A -85,B 0,C 180,E1 -3791.904,E2 -3791.904} C_VEL
LIN {X 0,Y 545.087,Z 352.587,A -85,B 0,C 180,E1 -3794.944,E2 -3794.944} C_VEL
LIN {X 0,Y 545.081,Z 352.586,A -85,B 0,C 180,E1 -3798.026,E2 -3798.026} C_VEL
LIN {X 0,Y 545.097,Z 352.589,A -85,B 0,C 180,E1 -3800.372,E2 -3800.372} C_VEL
LIN {X 0,Y 545.093,Z 352.59,A -85,B 0,C 180,E1 -3803.559,E2 -3803.559} C_VEL
LIN {X 0,Y 545.081,Z 352.585,A -85,B 0,C 180,E1 -3806.001,E2 -3806.001} C_VEL
LIN {X 0,Y 545.091,Z 352.589,A -85,B 0,C 180,E1 -3808.748,E2 -3808.748} C_VEL
LIN {X 0,Y 545.061,Z 352.591,A -85,B 0,C 180,E1 -3811.679,E2 -3811.679} C_VEL
LIN {X 0,Y 545.08,Z 352.586,A -85,B 0,C 180,E1 -3814.563,E2 -3814.563} C_VEL
LIN {X 0,Y 545.065,Z 352.592,A -85,B 0,C 180,E1 -3817.007,E2 -3817.007} C_VEL
LIN {X 0,Y 544.358,Z 352.677,A -85,B 0,C 180,E1 -3817.623,E2 -3817.623} C_VEL
LIN {X 0,Y 541.494,Z 353.038,A -85,B 0,C 180,E1 -3818.624,E2 -3818.624} C_VEL
LIN {X 0,Y 539.108,Z 353.332,A -85,B 0,C 180,E1 -3819.43,E2 -3819.43} C_VEL
LIN {X 0,Y 538.098,Z 353.458,A -85,B 0,C 180,E1 -3820.052,E2 -3820.052} C_VEL
LIN {X 0,Y 538.023,Z 353.464,A -85,B 0,C 180,E1 -3820.262,E2 -3820.262} C_VEL
LIN {X 0,Y 538.029,Z 353.465,A -85,B 0,C 180,E1 -3822.988,E2 -3822.988} C_VEL
LIN {X 0,Y 538.032,Z 353.464,A -85,B 0,C 180,E1 -3825.926,E2 -3825.926} C_VEL
LIN {X 0,Y 538.051,Z 353.461,A -85,B 0,C 180,E1 -3829.224,E2 -3829.224} C_VEL
LIN {X 0,Y 537.994,Z 353.474,A -85,B 0,C 180,E1 -3832.122,E2 -3832.122} C_VEL
LIN {X 0,Y 538.001,Z 353.469,A -85,B 0,C 180,E1 -3834.916,E2 -3834.916} C_VEL
LIN {X 0,Y 538.029,Z 353.464,A -85,B 0,C 180,E1 -3837.618,E2 -3837.618} C_VEL
LIN {X 0,Y 538.019,Z 353.469,A -85,B 0,C 180,E1 -3840.239,E2 -3840.239} C_VEL
LIN {X 0,Y 538.07,Z 353.459,A -85,B 0,C 180,E1 -3842.797,E2 -3842.797} C_VEL
LIN {X 0,Y 538.051,Z 353.466,A -85,B 0,C 180,E1 -3845.293,E2 -3845.293} C_VEL
LIN {X 0,Y 538.026,Z 353.469,A -85,B 0,C 180,E1 -3848.546,E2 -3848.546} C_VEL
LIN {X 0,Y 538.042,Z 353.462,A -85,B 0,C 180,E1 -3850.94,E2 -3850.94} C_VEL
LIN {X 0,Y 538.029,Z 353.466,A -85,B 0,C 180,E1 -3853.299,E2 -3853.299} C_VEL
LIN {X 0,Y 538.068,Z 353.463,A -85,B 0,C 180,E1 -3855.631,E2 -3855.631} C_VEL
LIN {X 0,Y 538.082,Z 353.463,A -85,B 0,C 180,E1 -3858.702,E2 -3858.702} C_VEL
LIN {X 0,Y 538.089,Z 353.458,A -85,B 0,C 180,E1 -3861.74,E2 -3861.74} C_VEL
LIN {X 0,Y 538.168,Z 353.447,A -85,B 0,C 180,E1 -3864.755,E2 -3864.755} C_VEL
LIN {X 0,Y 538.172,Z 353.447,A -85,B 0,C 180,E1 -3867.755,E2 -3867.755} C_VEL
LIN {X 0,Y 538.186,Z 353.446,A -85,B 0,C 180,E1 -3870.748,E2 -3870.748} C_VEL
LIN {X 0,Y 538.14,Z 353.449,A -85,B 0,C 180,E1 -3872.995,E2 -3872.995} C_VEL
LIN {X 0,Y 538.125,Z 353.453,A -85,B 0,C 180,E1 -3875.997,E2 -3875.997} C_VEL
LIN {X 0,Y 538.072,Z 353.462,A -85,B 0,C 180,E1 -3879.018,E2 -3879.018} C_VEL
LIN {X 0,Y 538.087,Z 353.463,A -85,B 0,C 180,E1 -3882.063,E2 -3882.063} C_VEL
LIN {X 0,Y 538.049,Z 353.464,A -85,B 0,C 180,E1 -3885.144,E2 -3885.144} C_VEL
LIN {X 0,Y 538.033,Z 353.465,A -85,B 0,C 180,E1 -3888.27,E2 -3888.27} C_VEL
LIN {X 0,Y 538.042,Z 353.466,A -85,B 0,C 180,E1 -3890.651,E2 -3890.651} C_VEL
LIN {X 0,Y 538.008,Z 353.47,A -85,B 0,C 180,E1 -3893.888,E2 -3893.888} C_VEL
LIN {X 0,Y 538.046,Z 353.461,A -85,B 0,C 180,E1 -3896.367,E2 -3896.367} C_VEL
LIN {X 0,Y 538.035,Z 353.468,A -85,B 0,C 180,E1 -3898.934,E2 -3898.934} C_VEL
LIN {X 0,Y 538.018,Z 353.469,A -85,B 0,C 180,E1 -3901.888,E2 -3901.888} C_VEL
LIN {X 0,Y 538.015,Z 353.465,A -85,B 0,C 180,E1 -3904.618,E2 -3904.618} C_VEL
LIN {X 0,Y 538.008,Z 353.473,A -85,B 0,C 180,E1 -3907.17,E2 -3907.17} C_VEL
LIN {X 0,Y 538.027,Z 353.465,A -85,B 0,C 180,E1 -3909.797,E2 -3909.797} C_VEL
LIN {X 0,Y 538.028,Z 353.465,A -85,B 0,C 180,E1 -3912.785,E2 -3912.785} C_VEL
LIN {X 0,Y 538.011,Z 353.468,A -85,B 0,C 180,E1 -3915.138,E2 -3915.138} C_VEL
LIN {X 0,Y 538.034,Z 353.463,A -85,B 0,C 180,E1 -3918.227,E2 -3918.227} C_VEL
LIN {X 0,Y 538.019,Z 353.466,A -85,B 0,C 180,E1 -3921.17,E2 -3921.17} C_VEL
LIN {X 0,Y 538.029,Z 353.467,A -85,B 0,C 180,E1 -3924.084,E2 -3924.084} C_VEL
LIN {X 0,Y 538.034,Z 353.464,A -85,B 0,C 180,E1 -3926.727,E2 -3926.727} C_VEL
LIN {X 0,Y 538.092,Z 353.523,A -85,B 0,C 180,E1 -3930.082,E2 -3930.082} C_VEL
LIN {X 0,Y 537.984,Z 359.562,A -85,B 0,C 180,E1 -3932.792,E2 -3932.792} C_VEL
LIN {X 0,Y 537.917,Z 365.233,A -85,B 0,C 180,E1 -3935.286,E2 -3935.286} C_VEL
LIN {X 0,Y 537.852,Z 371.305,A -85,B 0,C 180,E1 -3938.086,E2 -3938.086} C_VEL
LIN {X 0,Y 537.743,Z 377.589,A -85,B 0,C 180,E1 -3940.929,E2 -3940.929} C_VEL
LIN {X 0,Y 537.69,Z 382.897,A -85,B 0,C 180,E1 -3943.288,E2 -3943.288} C_VEL
LIN {X 0,Y 537.643,Z 388.22,A -85,B 0,C 180,E1 -3945.619,E2 -3945.619} C_VEL
LIN {X 0,Y 537.58,Z 395.34,A -85,B 0,C 180,E1 -3948.691,E2 -3948.691} C_VEL
LIN {X 0,Y 537.542,Z 402.483,A -85,B 0,C 180,E1 -3951.731,E2 -3951.731} C_VEL
LIN {X 0,Y 537.581,Z 403.712,A -85,B 0,C 180,E1 -3952.252,E2 -3952.252} C_VEL
LIN {X 0,Y 538.125,Z 412.547,A -85,B 0,C 180,E1 -3952.59,E2 -3952.59} C_VEL
LIN {X 0,Y 537.984,Z 421.622,A -85,B 0,C 180,E1 -3953.079,E2 -3953.079} C_VEL
LIN {X 0,Y 537.91,Z 430.056,A -85,B 0,C 180,E1 -3953.686,E2 -3953.686} C_VEL
LIN {X 0,Y 537.724,Z 437.219,A -85,B 0,C 180,E1 -3954.375,E2 -3954.375} C_VEL
LIN {X 0,Y 537.764,Z 443.334,A -85,B 0,C 180,E1 -3955.127,E2 -3955.127} C_VEL
LIN {X 0,Y 537.658,Z 448.158,A -85,B 0,C 180,E1 -3955.877,E2 -3955.877} C_VEL
LIN {X 0,Y 537.643,Z 451.872,A -85,B 0,C 180,E1 -3956.628,E2 -3956.628} C_VEL
LIN {X 0,Y 537.508,Z 455.848,A -85,B 0,C 180,E1 -3957.752,E2 -3957.752} C_VEL
LIN {X 0,Y 537.455,Z 457.586,A -85,B 0,C 180,E1 -3958.501,E2 -3958.501} C_VEL
LIN {X 0,Y 537.443,Z 458.625,A -85,B 0,C 180,E1 -3959.251,E2 -3959.251} C_VEL
LIN {X 0,Y 537.442,Z 458.996,A -85,B 0,C 180,E1 -3960,E2 -3960} C_VEL
LIN {X 0,Y 537.442,Z 458.708,A -85,B 0,C 180,E1 -3960.749,E2 -3960.749} C_VEL
LIN {X 0,Y 537.455,Z 457.756,A -85,B 0,C 180,E1 -3961.499,E2 -3961.499} C_VEL
LIN {X 0,Y 537.508,Z 456.118,A -85,B 0,C 180,E1 -3962.248,E2 -3962.248} C_VEL
LIN {X 0,Y 537.642,Z 452.247,A -85,B 0,C 180,E1 -3963.372,E2 -3963.372} C_VEL
LIN {X 0,Y 537.666,Z 447.608,A -85,B 0,C 180,E1 -3964.31,E2 -3964.31} C_VEL
LIN {X 0,Y 537.734,Z 442.648,A -85,B 0,C 180,E1 -3965.061,E2 -3965.061} C_VEL
LIN {X 0,Y 537.769,Z 436.394,A -85,B 0,C 180,E1 -3965.813,E2 -3965.813} C_VEL
LIN {X 0,Y 537.923,Z 429.684,A -85,B 0,C 180,E1 -3966.441,E2 -3966.441} C_VEL
LIN {X 0,Y 537.96,Z 421.533,A -85,B 0,C 180,E1 -3967.025,E2 -3967.025} C_VEL
LIN {X 0,Y 538.09,Z 412.641,A -85,B 0,C 180,E1 -3967.505,E2 -3967.505} C_VEL
LIN {X 0,Y 537.624,Z 404.564,A -85,B 0,C 180,E1 -3967.818,E2 -3967.818} C_VEL
LIN {X 0,Y 537.566,Z 403.837,A -85,B 0,C 180,E1 -3967.843,E2 -3967.843} C_VEL
LIN {X 0,Y 537.609,Z 395.849,A -85,B 0,C 180,E1 -3971.308,E2 -3971.308} C_VEL
LIN {X 0,Y 537.715,Z 388.174,A -85,B 0,C 180,E1 -3974.717,E2 -3974.717} C_VEL
LIN {X 0,Y 537.812,Z 382.076,A -85,B 0,C 180,E1 -3977.491,E2 -3977.491} C_VEL
LIN {X 0,Y 537.871,Z 376.967,A -85,B 0,C 180,E1 -3979.86,E2 -3979.86} C_VEL
LIN {X 0,Y 537.933,Z 371.507,A -85,B 0,C 180,E1 -3982.264,E2 -3982.264} C_VEL
LIN {X 0,Y 538.006,Z 366.169,A -85,B 0,C 180,E1 -3984.71,E2 -3984.71} C_VEL
LIN {X 0,Y 538.119,Z 360.212,A -85,B 0,C 180,E1 -3987.364,E2 -3987.364} C_VEL
LIN {X 0,Y 538.171,Z 353.573,A -85,B 0,C 180,E1 -3990.336,E2 -3990.336} C_VEL
LIN {X 0,Y 538.049,Z 353.466,A -85,B 0,C 180,E1 -3993.283,E2 -3993.283} C_VEL
LIN {X 0,Y 537.998,Z 353.474,A -85,B 0,C 180,E1 -3996.004,E2 -3996.004} C_VEL
LIN {X 0,Y 538.02,Z 353.47,A -85,B 0,C 180,E1 -3998.83,E2 -3998.83} C_VEL
LIN {X 0,Y 538.082,Z 353.462,A -85,B 0,C 180,E1 -4000.773,E2 -4000.773} C_VEL
LIN {X 0,Y 538.033,Z 353.468,A -85,B 0,C 180,E1 -4004.075,E2 -4004.075} C_VEL
LIN {X 0,Y 538.028,Z 353.469,A -85,B 0,C 180,E1 -4007.215,E2 -4007.215} C_VEL
LIN {X 0,Y 538.025,Z 353.469,A -85,B 0,C 180,E1 -4010.203,E2 -4010.203} C_VEL
LIN {X 0,Y 538.027,Z 353.469,A -85,B 0,C 180,E1 -4013.067,E2 -4013.067} C_VEL
LIN {X 0,Y 538.024,Z 353.471,A -85,B 0,C 180,E1 -4015.827,E2 -4015.827} C_VEL
LIN {X 0,Y 538.013,Z 353.473,A -85,B 0,C 180,E1 -4018.499,E2 -4018.499} C_VEL
LIN {X 0,Y 538.073,Z 353.634,A -85,B 0,C 180,E1 -4019.675,E2 -4019.675} C_VEL
LIN {X 0,Y 539.972,Z 362.18,A -85,B 0,C 180,E1 -4021.636,E2 -4021.636} C_VEL
LIN {X 0,Y 540.038,Z 366.79,A -85,B 0,C 180,E1 -4022.564,E2 -4022.564} C_VEL
LIN {X 0,Y 539.341,Z 383.205,A -85,B 0,C 180,E1 -4025.644,E2 -4025.644} C_VEL
LIN {X 0,Y 539.046,Z 395.257,A -85,B 0,C 180,E1 -4027.784,E2 -4027.784} C_VEL
LIN {X 0,Y 538.669,Z 411.558,A -85,B 0,C 180,E1 -4030.567,E2 -4030.567} C_VEL
LIN {X 0,Y 538.433,Z 428.058,A -85,B 0,C 180,E1 -4033.312,E2 -4033.312} C_VEL
LIN {X 0,Y 538.199,Z 444.518,A -85,B 0,C 180,E1 -4036.02,E2 -4036.02} C_VEL
LIN {X 0,Y 538.18,Z 448.188,A -85,B 0,C 180,E1 -4036.609,E2 -4036.609} C_VEL
LIN {X 0,Y 539.264,Z 457.218,A -85,B 0,C 180,E1 -4036.792,E2 -4036.792} C_VEL
LIN {X 0,Y 539.099,Z 470.496,A -85,B 0,C 180,E1 -4037.148,E2 -4037.148} C_VEL
LIN {X 0,Y 538.934,Z 482.506,A -85,B 0,C 180,E1 -4037.622,E2 -4037.622} C_VEL
LIN {X 0,Y 538.702,Z 494.637,A -85,B 0,C 180,E1 -4038.264,E2 -4038.264} C_VEL
LIN {X 0,Y 538.52,Z 505.483,A -85,B 0,C 180,E1 -4038.997,E2 -4038.997} C_VEL
LIN {X 0,Y 538.278,Z 515.644,A -85,B 0,C 180,E1 -4039.848,E2 -4039.848} C_VEL
LIN {X 0,Y 538.055,Z 524.784,A -85,B 0,C 180,E1 -4040.792,E2 -4040.792} C_VEL
LIN {X 0,Y 537.851,Z 533.687,A -85,B 0,C 180,E1 -4041.925,E2 -4041.925} C_VEL
LIN {X 0,Y 537.729,Z 540.848,A -85,B 0,C 180,E1 -4043.056,E2 -4043.056} C_VEL
LIN {X 0,Y 537.676,Z 547.365,A -85,B 0,C 180,E1 -4044.374,E2 -4044.374} C_VEL
LIN {X 0,Y 537.557,Z 551.676,A -85,B 0,C 180,E1 -4045.501,E2 -4045.501} C_VEL
LIN {X 0,Y 537.591,Z 553.958,A -85,B 0,C 180,E1 -4046.252,E2 -4046.252} C_VEL
LIN {X 0,Y 537.551,Z 555.807,A -85,B 0,C 180,E1 -4047.002,E2 -4047.002} C_VEL
LIN {X 0,Y 537.452,Z 558.183,A -85,B 0,C 180,E1 -4048.501,E2 -4048.501} C_VEL
LIN {X 0,Y 537.442,Z 559,A -85,B 0,C 180,E1 -4050,E2 -4050} C_VEL
LIN {X 0,Y 537.452,Z 558.184,A -85,B 0,C 180,E1 -4051.498,E2 -4051.498} C_VEL
LIN {X 0,Y 537.49,Z 557.197,A -85,B 0,C 180,E1 -4052.248,E2 -4052.248} C_VEL
LIN {X 0,Y 537.551,Z 555.81,A -85,B 0,C 180,E1 -4052.998,E2 -4052.998} C_VEL
LIN {X 0,Y 537.603,Z 552.897,A -85,B 0,C 180,E1 -4054.123,E2 -4054.123} C_VEL
LIN {X 0,Y 537.587,Z 548.95,A -85,B 0,C 180,E1 -4055.25,E2 -4055.25} C_VEL
LIN {X 0,Y 537.643,Z 544.131,A -85,B 0,C 180,E1 -4056.325,E2 -4056.325} C_VEL
LIN {X 0,Y 537.791,Z 537.466,A -85,B 0,C 180,E1 -4057.509,E2 -4057.509} C_VEL
LIN {X 0,Y 537.972,Z 529.478,A -85,B 0,C 180,E1 -4058.64,E2 -4058.64} C_VEL
LIN {X 0,Y 538.119,Z 521.334,A -85,B 0,C 180,E1 -4059.585,E2 -4059.585} C_VEL
LIN {X 0,Y 538.369,Z 511.4,A -85,B 0,C 180,E1 -4060.53,E2 -4060.53} C_VEL
LIN {X 0,Y 538.566,Z 501.592,A -85,B 0,C 180,E1 -4061.288,E2 -4061.288} C_VEL
LIN {X 0,Y 538.804,Z 490.702,A -85,B 0,C 180,E1 -4061.963,E2 -4061.963} C_VEL
LIN {X 0,Y 538.988,Z 478.104,A -85,B 0,C 180,E1 -4062.568,E2 -4062.568} C_VEL
LIN {X 0,Y 539.191,Z 465.089,A -85,B 0,C 180,E1 -4063.017,E2 -4063.017} C_VEL
LIN {X 0,Y 539.053,Z 454.334,A -85,B 0,C 180,E1 -4063.273,E2 -4063.273} C_VEL
LIN {X 0,Y 538.161,Z 447.982,A -85,B 0,C 180,E1 -4063.403,E2 -4063.403} C_VEL
LIN {X 0,Y 538.404,Z 430.514,A -85,B 0,C 180,E1 -4066.299,E2 -4066.299} C_VEL
LIN {X 0,Y 538.676,Z 412.85,A -85,B 0,C 180,E1 -4069.234,E2 -4069.234} C_VEL
LIN {X 0,Y 538.957,Z 400.141,A -85,B 0,C 180,E1 -4071.415,E2 -4071.415} C_VEL
LIN {X 0,Y 539.356,Z 385.131,A -85,B 0,C 180,E1 -4074.091,E2 -4074.091} C_VEL
LIN {X 0,Y 539.876,Z 368.277,A -85,B 0,C 180,E1 -4077.105,E2 -4077.105} C_VEL
LIN {X 0,Y 539.929,Z 362.536,A -85,B 0,C 180,E1 -4078.154,E2 -4078.154} C_VEL
LIN {X 0,Y 538.037,Z 353.469,A -85,B 0,C 180,E1 -4080.025,E2 -4080.025} C_VEL
LIN {X 0,Y 538.047,Z 353.466,A -85,B 0,C 180,E1 -4083.283,E2 -4083.283} C_VEL
LIN {X 0,Y 537.996,Z 353.468,A -85,B 0,C 180,E1 -4086.004,E2 -4086.004} C_VEL
LIN {X 0,Y 538.014,Z 353.468,A -85,B 0,C 180,E1 -4088.83,E2 -4088.83} C_VEL
LIN {X 0,Y 538.037,Z 353.469,A -85,B 0,C 180,E1 -4091.879,E2 -4091.879} C_VEL
LIN {X 0,Y 538.035,Z 353.468,A -85,B 0,C 180,E1 -4095.141,E2 -4095.141} C_VEL
LIN {X 0,Y 538.036,Z 353.466,A -85,B 0,C 180,E1 -4098.227,E2 -4098.227} C_VEL
LIN {X 0,Y 538.017,Z 353.465,A -85,B 0,C 180,E1 -4101.17,E2 -4101.17} C_VEL
LIN {X 0,Y 538.027,Z 353.465,A -85,B 0,C 180,E1 -4104.084,E2 -4104.084} C_VEL
LIN {X 0,Y 538.031,Z 353.469,A -85,B 0,C 180,E1 -4106.727,E2 -4106.727} C_VEL
LIN {X 0,Y 538.028,Z 353.464,A -85,B 0,C 180,E1 -4109.556,E2 -4109.556} C_VEL
LIN {X 0,Y 538.048,Z 353.467,A -85,B 0,C 180,E1 -4111.95,E2 -4111.95} C_VEL
LIN {X 0,Y 538.073,Z 353.458,A -85,B 0,C 180,E1 -4114.467,E2 -4114.467} C_VEL
LIN {X 0,Y 537.994,Z 353.468,A -85,B 0,C 180,E1 -4117.738,E2 -4117.738} C_VEL
LIN {X 0,Y 538.081,Z 353.463,A -85,B 0,C 180,E1 -4120.148,E2 -4120.148} C_VEL
LIN {X 0,Y 538.027,Z 353.466,A -85,B 0,C 180,E1 -4123.299,E2 -4123.299} C_VEL
LIN {X 0,Y 538.067,Z 353.461,A -85,B 0,C 180,E1 -4125.631,E2 -4125.631} C_VEL
LIN {X 0,Y 538.08,Z 353.462,A -85,B 0,C 180,E1 -4128.702,E2 -4128.702} C_VEL
LIN {X 0,Y 538.087,Z 353.461,A -85,B 0,C 180,E1 -4131.74,E2 -4131.74} C_VEL
LIN {X 0,Y 538.164,Z 353.448,A -85,B 0,C 180,E1 -4134.755,E2 -4134.755} C_VEL
LIN {X 0,Y 538.167,Z 353.447,A -85,B 0,C 180,E1 -4137.755,E2 -4137.755} C_VEL
LIN {X 0,Y 538.185,Z 353.446,A -85,B 0,C 180,E1 -4140.748,E2 -4140.748} C_VEL
LIN {X 0,Y 538.14,Z 353.45,A -85,B 0,C 180,E1 -4142.994,E2 -4142.994} C_VEL
LIN {X 0,Y 538.125,Z 353.452,A -85,B 0,C 180,E1 -4145.997,E2 -4145.997} C_VEL
LIN {X 0,Y 538.074,Z 353.46,A -85,B 0,C 180,E1 -4149.018,E2 -4149.018} C_VEL
LIN {X 0,Y 538.086,Z 353.461,A -85,B 0,C 180,E1 -4152.063,E2 -4152.063} C_VEL
LIN {X 0,Y 538.047,Z 353.466,A -85,B 0,C 180,E1 -4155.144,E2 -4155.144} C_VEL
LIN {X 0,Y 538.034,Z 353.466,A -85,B 0,C 180,E1 -4158.27,E2 -4158.27} C_VEL
LIN {X 0,Y 538.041,Z 353.465,A -85,B 0,C 180,E1 -4160.651,E2 -4160.651} C_VEL
LIN {X 0,Y 538.026,Z 353.467,A -85,B 0,C 180,E1 -4163.887,E2 -4163.887} C_VEL
LIN {X 0,Y 538.043,Z 353.462,A -85,B 0,C 180,E1 -4166.367,E2 -4166.367} C_VEL
LIN {X 0,Y 538.032,Z 353.466,A -85,B 0,C 180,E1 -4168.934,E2 -4168.934} C_VEL
LIN {X 0,Y 538.016,Z 353.47,A -85,B 0,C 180,E1 -4171.888,E2 -4171.888} C_VEL
LIN {X 0,Y 538.029,Z 353.464,A -85,B 0,C 180,E1 -4174.62,E2 -4174.62} C_VEL
LIN {X 0,Y 538.008,Z 353.47,A -85,B 0,C 180,E1 -4177.17,E2 -4177.17} C_VEL
LIN {X 0,Y 538.023,Z 353.464,A -85,B 0,C 180,E1 -4180.262,E2 -4180.262} C_VEL
LIN {X 0,Y 537.372,Z 353.548,A -85,B 0,C 180,E1 -4180.888,E2 -4180.888} C_VEL
LIN {X 0,Y 534.52,Z 353.909,A -85,B 0,C 180,E1 -4181.902,E2 -4181.902} C_VEL
LIN {X 0,Y 532.094,Z 354.213,A -85,B 0,C 180,E1 -4182.72,E2 -4182.72} C_VEL
LIN {X 0,Y 531.047,Z 354.34,A -85,B 0,C 180,E1 -4183.351,E2 -4183.351} C_VEL
LIN {X 0,Y 530.959,Z 354.349,A -85,B 0,C 180,E1 -4183.564,E2 -4183.564} C_VEL
LIN {X 0,Y 530.969,Z 354.344,A -85,B 0,C 180,E1 -4186.506,E2 -4186.506} C_VEL
LIN {X 0,Y 530.984,Z 354.341,A -85,B 0,C 180,E1 -4189.567,E2 -4189.567} C_VEL
LIN {X 0,Y 530.97,Z 354.344,A -85,B 0,C 180,E1 -4192.577,E2 -4192.577} C_VEL
LIN {X 0,Y 530.985,Z 354.346,A -85,B 0,C 180,E1 -4195.31,E2 -4195.31} C_VEL
LIN {X 0,Y 530.974,Z 354.343,A -85,B 0,C 180,E1 -4198.032,E2 -4198.032} C_VEL
LIN {X 0,Y 530.992,Z 354.341,A -85,B 0,C 180,E1 -4200.874,E2 -4200.874} C_VEL
LIN {X 0,Y 531.009,Z 354.34,A -85,B 0,C 180,E1 -4203.257,E2 -4203.257} C_VEL
LIN {X 0,Y 530.988,Z 354.342,A -85,B 0,C 180,E1 -4205.961,E2 -4205.961} C_VEL
LIN {X 0,Y 531.003,Z 354.341,A -85,B 0,C 180,E1 -4209.062,E2 -4209.062} C_VEL
LIN {X 0,Y 531.02,Z 354.34,A -85,B 0,C 180,E1 -4212.278,E2 -4212.278} C_VEL
LIN {X 0,Y 531.023,Z 354.341,A -85,B 0,C 180,E1 -4215.436,E2 -4215.436} C_VEL
LIN {X 0,Y 531.041,Z 354.339,A -85,B 0,C 180,E1 -4218.55,E2 -4218.55} C_VEL
LIN {X 0,Y 531.058,Z 354.333,A -85,B 0,C 180,E1 -4221.63,E2 -4221.63} C_VEL
LIN {X 0,Y 531.126,Z 354.324,A -85,B 0,C 180,E1 -4224.685,E2 -4224.685} C_VEL
LIN {X 0,Y 531.144,Z 354.322,A -85,B 0,C 180,E1 -4227.725,E2 -4227.725} C_VEL
LIN {X 0,Y 531.157,Z 354.322,A -85,B 0,C 180,E1 -4230.758,E2 -4230.758} C_VEL
LIN {X 0,Y 531.107,Z 354.325,A -85,B 0,C 180,E1 -4233.034,E2 -4233.034} C_VEL
LIN {X 0,Y 531.08,Z 354.33,A -85,B 0,C 180,E1 -4236.077,E2 -4236.077} C_VEL
LIN {X 0,Y 531.059,Z 354.335,A -85,B 0,C 180,E1 -4238.371,E2 -4238.371} C_VEL
LIN {X 0,Y 531.056,Z 354.334,A -85,B 0,C 180,E1 -4241.672,E2 -4241.672} C_VEL
LIN {X 0,Y 531.035,Z 354.336,A -85,B 0,C 180,E1 -4244.956,E2 -4244.956} C_VEL
LIN {X 0,Y 531.021,Z 354.338,A -85,B 0,C 180,E1 -4247.722,E2 -4247.722} C_VEL
LIN {X 0,Y 531.003,Z 354.34,A -85,B 0,C 180,E1 -4250.938,E2 -4250.938} C_VEL
LIN {X 0,Y 530.97,Z 354.343,A -85,B 0,C 180,E1 -4254.225,E2 -4254.225} C_VEL
LIN {X 0,Y 531.009,Z 354.34,A -85,B 0,C 180,E1 -4256.744,E2 -4256.744} C_VEL
LIN {X 0,Y 530.986,Z 354.342,A -85,B 0,C 180,E1 -4259.323,E2 -4259.323} C_VEL
LIN {X 0,Y 530.974,Z 354.348,A -85,B 0,C 180,E1 -4262.101,E2 -4262.101} C_VEL
LIN {X 0,Y 530.974,Z 354.343,A -85,B 0,C 180,E1 -4264.851,E2 -4264.851} C_VEL
LIN {X 0,Y 530.969,Z 354.345,A -85,B 0,C 180,E1 -4267.508,E2 -4267.508} C_VEL
LIN {X 0,Y 530.985,Z 354.346,A -85,B 0,C 180,E1 -4270.433,E2 -4270.433} C_VEL
LIN {X 0,Y 530.974,Z 354.344,A -85,B 0,C 180,E1 -4273.282,E2 -4273.282} C_VEL
LIN {X 0,Y 530.98,Z 354.345,A -85,B 0,C 180,E1 -4275.622,E2 -4275.622} C_VEL
LIN {X 0,Y 530.997,Z 354.343,A -85,B 0,C 180,E1 -4278.564,E2 -4278.564} C_VEL
LIN {X 0,Y 530.963,Z 354.345,A -85,B 0,C 180,E1 -4281.53,E2 -4281.53} C_VEL
LIN {X 0,Y 530.981,Z 354.343,A -85,B 0,C 180,E1 -4284.382,E2 -4284.382} C_VEL
LIN {X 0,Y 530.971,Z 354.349,A -85,B 0,C 180,E1 -4287.133,E2 -4287.133} C_VEL
LIN {X 0,Y 531.077,Z 354.361,A -85,B 0,C 180,E1 -4290.029,E2 -4290.029} C_VEL
LIN {X 0,Y 530.926,Z 361.445,A -85,B 0,C 180,E1 -4293.252,E2 -4293.252} C_VEL
LIN {X 0,Y 530.862,Z 367.604,A -85,B 0,C 180,E1 -4295.991,E2 -4295.991} C_VEL
LIN {X 0,Y 530.735,Z 374.174,A -85,B 0,C 180,E1 -4299.051,E2 -4299.051} C_VEL
LIN {X 0,Y 530.683,Z 379.471,A -85,B 0,C 180,E1 -4301.468,E2 -4301.468} C_VEL
LIN {X 0,Y 530.597,Z 384.784,A -85,B 0,C 180,E1 -4303.85,E2 -4303.85} C_VEL
LIN {X 0,Y 530.526,Z 390.111,A -85,B 0,C 180,E1 -4306.205,E2 -4306.205} C_VEL
LIN {X 0,Y 530.471,Z 397.235,A -85,B 0,C 180,E1 -4309.311,E2 -4309.311} C_VEL
LIN {X 0,Y 530.481,Z 403.892,A -85,B 0,C 180,E1 -4312.123,E2 -4312.123} C_VEL
LIN {X 0,Y 531.111,Z 412.376,A -85,B 0,C 180,E1 -4312.449,E2 -4312.449} C_VEL
LIN {X 0,Y 530.989,Z 420.964,A -85,B 0,C 180,E1 -4312.901,E2 -4312.901} C_VEL
LIN {X 0,Y 530.927,Z 428.257,A -85,B 0,C 180,E1 -4313.41,E2 -4313.41} C_VEL
LIN {X 0,Y 530.734,Z 436.1,A -85,B 0,C 180,E1 -4314.11,E2 -4314.11} C_VEL
LIN {X 0,Y 530.697,Z 442.549,A -85,B 0,C 180,E1 -4314.871,E2 -4314.871} C_VEL
LIN {X 0,Y 530.631,Z 447.64,A -85,B 0,C 180,E1 -4315.632,E2 -4315.632} C_VEL
LIN {X 0,Y 530.611,Z 452.504,A -85,B 0,C 180,E1 -4316.583,E2 -4316.583} C_VEL
LIN {X 0,Y 530.444,Z 456.495,A -85,B 0,C 180,E1 -4317.722,E2 -4317.722} C_VEL
LIN {X 0,Y 530.388,Z 458.231,A -85,B 0,C 180,E1 -4318.481,E2 -4318.481} C_VEL
LIN {X 0,Y 530.374,Z 459.271,A -85,B 0,C 180,E1 -4319.241,E2 -4319.241} C_VEL
LIN {X 0,Y 530.373,Z 459.648,A -85,B 0,C 180,E1 -4320,E2 -4320} C_VEL
LIN {X 0,Y 530.375,Z 459.372,A -85,B 0,C 180,E1 -4320.759,E2 -4320.759} C_VEL
LIN {X 0,Y 530.391,Z 458.437,A -85,B 0,C 180,E1 -4321.519,E2 -4321.519} C_VEL
LIN {X 0,Y 530.508,Z 455.693,A -85,B 0,C 180,E1 -4322.658,E2 -4322.658} C_VEL
LIN {X 0,Y 530.609,Z 452.957,A -85,B 0,C 180,E1 -4323.417,E2 -4323.417} C_VEL
LIN {X 0,Y 530.63,Z 448.33,A -85,B 0,C 180,E1 -4324.368,E2 -4324.368} C_VEL
LIN {X 0,Y 530.705,Z 443.389,A -85,B 0,C 180,E1 -4325.128,E2 -4325.128} C_VEL
LIN {X 0,Y 530.754,Z 437.155,A -85,B 0,C 180,E1 -4325.89,E2 -4325.89} C_VEL
LIN {X 0,Y 530.953,Z 429.664,A -85,B 0,C 180,E1 -4326.593,E2 -4326.593} C_VEL
LIN {X 0,Y 530.967,Z 422.452,A -85,B 0,C 180,E1 -4327.118,E2 -4327.118} C_VEL
LIN {X 0,Y 531.131,Z 412.697,A -85,B 0,C 180,E1 -4327.652,E2 -4327.652} C_VEL
LIN {X 0,Y 530.518,Z 404.255,A -85,B 0,C 180,E1 -4327.996,E2 -4327.996} C_VEL
LIN {X 0,Y 530.558,Z 396.272,A -85,B 0,C 180,E1 -4331.461,E2 -4331.461} C_VEL
LIN {X 0,Y 530.67,Z 388.781,A -85,B 0,C 180,E1 -4334.808,E2 -4334.808} C_VEL
LIN {X 0,Y 530.772,Z 382.442,A -85,B 0,C 180,E1 -4337.731,E2 -4337.731} C_VEL
LIN {X 0,Y 530.831,Z 377.2,A -85,B 0,C 180,E1 -4340.135,E2 -4340.135} C_VEL
LIN {X 0,Y 530.918,Z 371.858,A -85,B 0,C 180,E1 -4342.575,E2 -4342.575} C_VEL
LIN {X 0,Y 531.008,Z 366.434,A -85,B 0,C 180,E1 -4345.058,E2 -4345.058} C_VEL
LIN {X 0,Y 531.109,Z 360.856,A -85,B 0,C 180,E1 -4347.59,E2 -4347.59} C_VEL
LIN {X 0,Y 531.234,Z 355.163,A -85,B 0,C 180,E1 -4350.18,E2 -4350.18} C_VEL
LIN {X 0,Y 531.068,Z 354.338,A -85,B 0,C 180,E1 -4350.661,E2 -4350.661} C_VEL
LIN {X 0,Y 530.991,Z 354.347,A -85,B 0,C 180,E1 -4353.773,E2 -4353.773} C_VEL
LIN {X 0,Y 530.959,Z 354.349,A -85,B 0,C 180,E1 -4356.558,E2 -4356.558} C_VEL
LIN {X 0,Y 531.01,Z 354.343,A -85,B 0,C 180,E1 -4359.857,E2 -4359.857} C_VEL
LIN {X 0,Y 530.987,Z 354.346,A -85,B 0,C 180,E1 -4362.456,E2 -4362.456} C_VEL
LIN {X 0,Y 530.992,Z 354.345,A -85,B 0,C 180,E1 -4365.621,E2 -4365.621} C_VEL
LIN {X 0,Y 531.001,Z 354.345,A -85,B 0,C 180,E1 -4368.565,E2 -4368.565} C_VEL
LIN {X 0,Y 530.959,Z 354.35,A -85,B 0,C 180,E1 -4371.529,E2 -4371.529} C_VEL
LIN {X 0,Y 530.958,Z 354.349,A -85,B 0,C 180,E1 -4374.38,E2 -4374.38} C_VEL
LIN {X 0,Y 530.974,Z 354.351,A -85,B 0,C 180,E1 -4377.134,E2 -4377.134} C_VEL
LIN {X 0,Y 530.973,Z 354.36,A -85,B 0,C 180,E1 -4379.267,E2 -4379.267} C_VEL
LIN {X 0,Y 533.03,Z 363.505,A -85,B 0,C 180,E1 -4381.448,E2 -4381.448} C_VEL
LIN {X 0,Y 533.224,Z 367.305,A -85,B 0,C 180,E1 -4382.265,E2 -4382.265} C_VEL
LIN {X 0,Y 532.521,Z 381.621,A -85,B 0,C 180,E1 -4385.018,E2 -4385.018} C_VEL
LIN {X 0,Y 532.075,Z 395.743,A -85,B 0,C 180,E1 -4387.61,E2 -4387.61} C_VEL
LIN {X 0,Y 531.671,Z 413.475,A -85,B 0,C 180,E1 -4390.703,E2 -4390.703} C_VEL
LIN {X 0,Y 531.399,Z 429.927,A -85,B 0,C 180,E1 -4393.48,E2 -4393.48} C_VEL
LIN {X 0,Y 531.12,Z 447.858,A -85,B 0,C 180,E1 -4396.44,E2 -4396.44} C_VEL
LIN {X 0,Y 532.326,Z 457.647,A -85,B 0,C 180,E1 -4396.641,E2 -4396.641} C_VEL
LIN {X 0,Y 532.196,Z 470.129,A -85,B 0,C 180,E1 -4396.978,E2 -4396.978} C_VEL
LIN {X 0,Y 532,Z 482.385,A -85,B 0,C 180,E1 -4397.458,E2 -4397.458} C_VEL
LIN {X 0,Y 531.752,Z 493.558,A -85,B 0,C 180,E1 -4398.044,E2 -4398.044} C_VEL
LIN {X 0,Y 531.538,Z 505.481,A -85,B 0,C 180,E1 -4398.85,E2 -4398.85} C_VEL
LIN {X 0,Y 531.263,Z 515.644,A -85,B 0,C 180,E1 -4399.712,E2 -4399.712} C_VEL
LIN {X 0,Y 531.012,Z 524.784,A -85,B 0,C 180,E1 -4400.669,E2 -4400.669} C_VEL
LIN {X 0,Y 530.813,Z 533.686,A -85,B 0,C 180,E1 -4401.817,E2 -4401.817} C_VEL
LIN {X 0,Y 530.664,Z 540.847,A -85,B 0,C 180,E1 -4402.963,E2 -4402.963} C_VEL
LIN {X 0,Y 530.611,Z 547.365,A -85,B 0,C 180,E1 -4404.299,E2 -4404.299} C_VEL
LIN {X 0,Y 530.457,Z 551.676,A -85,B 0,C 180,E1 -4405.44,E2 -4405.44} C_VEL
LIN {X 0,Y 530.516,Z 553.957,A -85,B 0,C 180,E1 -4406.202,E2 -4406.202} C_VEL
LIN {X 0,Y 530.457,Z 555.806,A -85,B 0,C 180,E1 -4406.962,E2 -4406.962} C_VEL
LIN {X 0,Y 530.411,Z 557.193,A -85,B 0,C 180,E1 -4407.722,E2 -4407.722} C_VEL
LIN {X 0,Y 530.344,Z 558.785,A -85,B 0,C 180,E1 -4409.241,E2 -4409.241} C_VEL
LIN {X 0,Y 530.342,Z 559,A -85,B 0,C 180,E1 -4410,E2 -4410} C_VEL
LIN {X 0,Y 530.361,Z 558.184,A -85,B 0,C 180,E1 -4411.519,E2 -4411.519} C_VEL
LIN {X 0,Y 530.411,Z 557.197,A -85,B 0,C 180,E1 -4412.278,E2 -4412.278} C_VEL
LIN {X 0,Y 530.457,Z 555.81,A -85,B 0,C 180,E1 -4413.038,E2 -4413.038} C_VEL
LIN {X 0,Y 530.522,Z 552.897,A -85,B 0,C 180,E1 -4414.178,E2 -4414.178} C_VEL
LIN {X 0,Y 530.524,Z 548.95,A -85,B 0,C 180,E1 -4415.321,E2 -4415.321} C_VEL
LIN {X 0,Y 530.595,Z 543.28,A -85,B 0,C 180,E1 -4416.578,E2 -4416.578} C_VEL
LIN {X 0,Y 530.758,Z 536.236,A -85,B 0,C 180,E1 -4417.8,E2 -4417.8} C_VEL
LIN {X 0,Y 530.931,Z 527.995,A -85,B 0,C 180,E1 -4418.948,E2 -4418.948} C_VEL
LIN {X 0,Y 531.119,Z 519.541,A -85,B 0,C 180,E1 -4419.905,E2 -4419.905} C_VEL
LIN {X 0,Y 531.423,Z 509.091,A -85,B 0,C 180,E1 -4420.862,E2 -4420.862} C_VEL
LIN {X 0,Y 531.665,Z 498.135,A -85,B 0,C 180,E1 -4421.671,E2 -4421.671} C_VEL
LIN {X 0,Y 531.91,Z 487.345,A -85,B 0,C 180,E1 -4422.301,E2 -4422.301} C_VEL
LIN {X 0,Y 532.085,Z 475.517,A -85,B 0,C 180,E1 -4422.83,E2 -4422.83} C_VEL
LIN {X 0,Y 532.305,Z 461.851,A -85,B 0,C 180,E1 -4423.262,E2 -4423.262} C_VEL
LIN {X 0,Y 532.164,Z 455.362,A -85,B 0,C 180,E1 -4423.411,E2 -4423.411} C_VEL
LIN {X 0,Y 531.108,Z 447.8,A -85,B 0,C 180,E1 -4423.584,E2 -4423.584} C_VEL
LIN {X 0,Y 531.4,Z 430.196,A -85,B 0,C 180,E1 -4426.52,E2 -4426.52} C_VEL
LIN {X 0,Y 531.699,Z 411.346,A -85,B 0,C 180,E1 -4429.698,E2 -4429.698} C_VEL
LIN {X 0,Y 531.98,Z 399.965,A -85,B 0,C 180,E1 -4431.71,E2 -4431.71} C_VEL
LIN {X 0,Y 532.413,Z 386.517,A -85,B 0,C 180,E1 -4434.155,E2 -4434.155} C_VEL
LIN {X 0,Y 533.008,Z 369.315,A -85,B 0,C 180,E1 -4437.271,E2 -4437.271} C_VEL
LIN {X 0,Y 532.981,Z 363.572,A -85,B 0,C 180,E1 -4438.34,E2 -4438.34} C_VEL
LIN {X 0,Y 530.997,Z 354.345,A -85,B 0,C 180,E1 -4440.312,E2 -4440.312} C_VEL
LIN {X 0,Y 531.001,Z 354.345,A -85,B 0,C 180,E1 -4443.506,E2 -4443.506} C_VEL
LIN {X 0,Y 530.957,Z 354.349,A -85,B 0,C 180,E1 -4446.558,E2 -4446.558} C_VEL
LIN {X 0,Y 530.987,Z 354.341,A -85,B 0,C 180,E1 -4449.443,E2 -4449.443} C_VEL
LIN {X 0,Y 530.984,Z 354.342,A -85,B 0,C 180,E1 -4452.456,E2 -4452.456} C_VEL
LIN {X 0,Y 530.99,Z 354.343,A -85,B 0,C 180,E1 -4455.621,E2 -4455.621} C_VEL
LIN {X 0,Y 530.998,Z 354.344,A -85,B 0,C 180,E1 -4458.565,E2 -4458.565} C_VEL
LIN {X 0,Y 530.961,Z 354.346,A -85,B 0,C 180,E1 -4461.53,E2 -4461.53} C_VEL
LIN {X 0,Y 530.979,Z 354.342,A -85,B 0,C 180,E1 -4464.382,E2 -4464.382} C_VEL
LIN {X 0,Y 530.969,Z 354.347,A -85,B 0,C 180,E1 -4467.133,E2 -4467.133} C_VEL
LIN {X 0,Y 530.972,Z 354.345,A -85,B 0,C 180,E1 -4469.803,E2 -4469.803} C_VEL
LIN {X 0,Y 531.018,Z 354.337,A -85,B 0,C 180,E1 -4472.467,E2 -4472.467} C_VEL
LIN {X 0,Y 531.007,Z 354.342,A -85,B 0,C 180,E1 -4474.942,E2 -4474.942} C_VEL
LIN {X 0,Y 530.973,Z 354.346,A -85,B 0,C 180,E1 -4478.247,E2 -4478.247} C_VEL
LIN {X 0,Y 530.996,Z 354.341,A -85,B 0,C 180,E1 -4480.677,E2 -4480.677} C_VEL
LIN {X 0,Y 530.988,Z 354.341,A -85,B 0,C 180,E1 -4483.071,E2 -4483.071} C_VEL
LIN {X 0,Y 531.043,Z 354.338,A -85,B 0,C 180,E1 -4485.436,E2 -4485.436} C_VEL
LIN {X 0,Y 531.039,Z 354.339,A -85,B 0,C 180,E1 -4488.55,E2 -4488.55} C_VEL
LIN {X 0,Y 531.057,Z 354.335,A -85,B 0,C 180,E1 -4491.629,E2 -4491.629} C_VEL
LIN {X 0,Y 531.123,Z 354.324,A -85,B 0,C 180,E1 -4494.685,E2 -4494.685} C_VEL
LIN {X 0,Y 531.139,Z 354.322,A -85,B 0,C 180,E1 -4497.725,E2 -4497.725} C_VEL
LIN {X 0,Y 531.155,Z 354.321,A -85,B 0,C 180,E1 -4500.758,E2 -4500.758} C_VEL
LIN {X 0,Y 531.107,Z 354.327,A -85,B 0,C 180,E1 -4503.034,E2 -4503.034} C_VEL
LIN {X 0,Y 531.085,Z 354.328,A -85,B 0,C 180,E1 -4506.077,E2 -4506.077} C_VEL
LIN {X 0,Y 531.034,Z 354.337,A -85,B 0,C 180,E1 -4509.138,E2 -4509.138} C_VEL
LIN {X 0,Y 531.043,Z 354.337,A -85,B 0,C 180,E1 -4512.225,E2 -4512.225} C_VEL
LIN {X 0,Y 530.997,Z 354.345,A -85,B 0,C 180,E1 -4515.35,E2 -4515.35} C_VEL
LIN {X 0,Y 530.993,Z 354.344,A -85,B 0,C 180,E1 -4518.521,E2 -4518.521} C_VEL
LIN {X 0,Y 531.002,Z 354.34,A -85,B 0,C 180,E1 -4520.938,E2 -4520.938} C_VEL
LIN {X 0,Y 530.982,Z 354.342,A -85,B 0,C 180,E1 -4524.225,E2 -4524.225} C_VEL
LIN {X 0,Y 531.003,Z 354.342,A -85,B 0,C 180,E1 -4526.744,E2 -4526.744} C_VEL
LIN {X 0,Y 530.983,Z 354.342,A -85,B 0,C 180,E1 -4529.323,E2 -4529.323} C_VEL
LIN {X 0,Y 530.972,Z 354.348,A -85,B 0,C 180,E1 -4532.101,E2 -4532.101} C_VEL
LIN {X 0,Y 530.985,Z 354.343,A -85,B 0,C 180,E1 -4534.853,E2 -4534.853} C_VEL
LIN {X 0,Y 530.968,Z 354.343,A -85,B 0,C 180,E1 -4537.508,E2 -4537.508} C_VEL
LIN {X 0,Y 530.986,Z 354.347,A -85,B 0,C 180,E1 -4540.433,E2 -4540.433} C_VEL
LIN {X 0,Y 530.966,Z 354.346,A -85,B 0,C 180,E1 -4543.282,E2 -4543.282} C_VEL
LIN {X 0,Y 530.959,Z 354.349,A -85,B 0,C 180,E1 -4543.564,E2 -4543.564} C_VEL
LIN {X 0,Y 530.289,Z 354.43,A -85,B 0,C 180,E1 -4544.198,E2 -4544.198} C_VEL
LIN {X 0,Y 527.445,Z 354.788,A -85,B 0,C 180,E1 -4545.227,E2 -4545.227} C_VEL
LIN {X 0,Y 525.044,Z 355.09,A -85,B 0,C 180,E1 -4546.055,E2 -4546.055} C_VEL
LIN {X 0,Y 524.01,Z 355.216,A -85,B 0,C 180,E1 -4546.695,E2 -4546.695} C_VEL
LIN {X 0,Y 523.925,Z 355.224,A -85,B 0,C 180,E1 -4546.911,E2 -4546.911} C_VEL
LIN {X 0,Y 523.95,Z 355.219,A -85,B 0,C 180,E1 -4549.921,E2 -4549.921} C_VEL
LIN {X 0,Y 523.909,Z 355.223,A -85,B 0,C 180,E1 -4552.868,E2 -4552.868} C_VEL
LIN {X 0,Y 523.935,Z 355.222,A -85,B 0,C 180,E1 -4555.71,E2 -4555.71} C_VEL
LIN {X 0,Y 523.926,Z 355.224,A -85,B 0,C 180,E1 -4558.456,E2 -4558.456} C_VEL
LIN {X 0,Y 523.942,Z 355.218,A -85,B 0,C 180,E1 -4561.126,E2 -4561.126} C_VEL
LIN {X 0,Y 523.987,Z 355.216,A -85,B 0,C 180,E1 -4563.98,E2 -4563.98} C_VEL
LIN {X 0,Y 523.929,Z 355.221,A -85,B 0,C 180,E1 -4566.27,E2 -4566.27} C_VEL
LIN {X 0,Y 523.949,Z 355.222,A -85,B 0,C 180,E1 -4568.767,E2 -4568.767} C_VEL
LIN {X 0,Y 523.956,Z 355.216,A -85,B 0,C 180,E1 -4571.221,E2 -4571.221} C_VEL
LIN {X 0,Y 523.941,Z 355.223,A -85,B 0,C 180,E1 -4573.639,E2 -4573.639} C_VEL
LIN {X 0,Y 523.943,Z 355.219,A -85,B 0,C 180,E1 -4576.028,E2 -4576.028} C_VEL
LIN {X 0,Y 524.016,Z 355.212,A -85,B 0,C 180,E1 -4578.394,E2 -4578.394} C_VEL
LIN {X 0,Y 524.007,Z 355.21,A -85,B 0,C 180,E1 -4581.516,E2 -4581.516} C_VEL
LIN {X 0,Y 524.086,Z 355.201,A -85,B 0,C 180,E1 -4584.614,E2 -4584.614} C_VEL
LIN {X 0,Y 524.116,Z 355.198,A -85,B 0,C 180,E1 -4587.695,E2 -4587.695} C_VEL
LIN {X 0,Y 524.127,Z 355.197,A -85,B 0,C 180,E1 -4590.768,E2 -4590.768} C_VEL
LIN {X 0,Y 524.074,Z 355.201,A -85,B 0,C 180,E1 -4593.075,E2 -4593.075} C_VEL
LIN {X 0,Y 524.041,Z 355.207,A -85,B 0,C 180,E1 -4596.159,E2 -4596.159} C_VEL
LIN {X 0,Y 524.008,Z 355.214,A -85,B 0,C 180,E1 -4598.484,E2 -4598.484} C_VEL
LIN {X 0,Y 524.007,Z 355.213,A -85,B 0,C 180,E1 -4601.74,E2 -4601.74} C_VEL
LIN {X 0,Y 523.997,Z 355.213,A -85,B 0,C 180,E1 -4605.052,E2 -4605.052} C_VEL
LIN {X 0,Y 523.967,Z 355.216,A -85,B 0,C 180,E1 -4607.969,E2 -4607.969} C_VEL
LIN {X 0,Y 523.976,Z 355.219,A -85,B 0,C 180,E1 -4610.41,E2 -4610.41} C_VEL
LIN {X 0,Y 523.915,Z 355.222,A -85,B 0,C 180,E1 -4612.894,E2 -4612.894} C_VEL
LIN {X 0,Y 523.988,Z 355.213,A -85,B 0,C 180,E1 -4616.02,E2 -4616.02} C_VEL
LIN {X 0,Y 523.944,Z 355.223,A -85,B 0,C 180,E1 -4618.875,E2 -4618.875} C_VEL
LIN {X 0,Y 523.927,Z 355.222,A -85,B 0,C 180,E1 -4621.544,E2 -4621.544} C_VEL
LIN {X 0,Y 523.936,Z 355.22,A -85,B 0,C 180,E1 -4624.29,E2 -4624.29} C_VEL
LIN {X 0,Y 523.911,Z 355.228,A -85,B 0,C 180,E1 -4627.132,E2 -4627.132} C_VEL
LIN {X 0,Y 523.941,Z 355.222,A -85,B 0,C 180,E1 -4630.13,E2 -4630.13} C_VEL
LIN {X 0,Y 523.943,Z 355.221,A -85,B 0,C 180,E1 -4632.459,E2 -4632.459} C_VEL
LIN {X 0,Y 523.947,Z 355.222,A -85,B 0,C 180,E1 -4635.31,E2 -4635.31} C_VEL
LIN {X 0,Y 523.959,Z 355.22,A -85,B 0,C 180,E1 -4638.69,E2 -4638.69} C_VEL
LIN {X 0,Y 523.923,Z 355.222,A -85,B 0,C 180,E1 -4641.08,E2 -4641.08} C_VEL
LIN {X 0,Y 523.929,Z 355.225,A -85,B 0,C 180,E1 -4643.827,E2 -4643.827} C_VEL
LIN {X 0,Y 523.945,Z 355.219,A -85,B 0,C 180,E1 -4646.636,E2 -4646.636} C_VEL
LIN {X 0,Y 524.06,Z 355.32,A -85,B 0,C 180,E1 -4650.03,E2 -4650.03} C_VEL
LIN {X 0,Y 523.859,Z 361.448,A -85,B 0,C 180,E1 -4652.862,E2 -4652.862} C_VEL
LIN {X 0,Y 523.81,Z 367.131,A -85,B 0,C 180,E1 -4655.422,E2 -4655.422} C_VEL
LIN {X 0,Y 523.727,Z 372.529,A -85,B 0,C 180,E1 -4657.93,E2 -4657.93} C_VEL
LIN {X 0,Y 523.658,Z 377.819,A -85,B 0,C 180,E1 -4660.396,E2 -4660.396} C_VEL
LIN {X 0,Y 523.573,Z 383.125,A -85,B 0,C 180,E1 -4662.824,E2 -4662.824} C_VEL
LIN {X 0,Y 523.468,Z 390.223,A -85,B 0,C 180,E1 -4666.015,E2 -4666.015} C_VEL
LIN {X 0,Y 523.395,Z 397.439,A -85,B 0,C 180,E1 -4669.165,E2 -4669.165} C_VEL
LIN {X 0,Y 523.395,Z 404.187,A -85,B 0,C 180,E1 -4671.992,E2 -4671.992} C_VEL
LIN {X 0,Y 524.115,Z 413.069,A -85,B 0,C 180,E1 -4672.342,E2 -4672.342} C_VEL
LIN {X 0,Y 523.98,Z 422.689,A -85,B 0,C 180,E1 -4672.873,E2 -4672.873} C_VEL
LIN {X 0,Y 523.862,Z 430.71,A -85,B 0,C 180,E1 -4673.466,E2 -4673.466} C_VEL
LIN {X 0,Y 523.673,Z 438.45,A -85,B 0,C 180,E1 -4674.223,E2 -4674.223} C_VEL
LIN {X 0,Y 523.704,Z 444.562,A -85,B 0,C 180,E1 -4674.996,E2 -4674.996} C_VEL
LIN {X 0,Y 523.581,Z 449.387,A -85,B 0,C 180,E1 -4675.766,E2 -4675.766} C_VEL
LIN {X 0,Y 523.579,Z 453.133,A -85,B 0,C 180,E1 -4676.537,E2 -4676.537} C_VEL
LIN {X 0,Y 523.381,Z 457.143,A -85,B 0,C 180,E1 -4677.691,E2 -4677.691} C_VEL
LIN {X 0,Y 523.322,Z 458.89,A -85,B 0,C 180,E1 -4678.461,E2 -4678.461} C_VEL
LIN {X 0,Y 523.307,Z 459.941,A -85,B 0,C 180,E1 -4679.23,E2 -4679.23} C_VEL
LIN {X 0,Y 523.306,Z 460.327,A -85,B 0,C 180,E1 -4680,E2 -4680} C_VEL
LIN {X 0,Y 523.31,Z 460.058,A -85,B 0,C 180,E1 -4680.769,E2 -4680.769} C_VEL
LIN {X 0,Y 523.328,Z 459.128,A -85,B 0,C 180,E1 -4681.539,E2 -4681.539} C_VEL
LIN {X 0,Y 523.465,Z 456.398,A -85,B 0,C 180,E1 -4682.693,E2 -4682.693} C_VEL
LIN {X 0,Y 523.576,Z 453.667,A -85,B 0,C 180,E1 -4683.463,E2 -4683.463} C_VEL
LIN {X 0,Y 523.595,Z 449.045,A -85,B 0,C 180,E1 -4684.426,E2 -4684.426} C_VEL
LIN {X 0,Y 523.681,Z 444.13,A -85,B 0,C 180,E1 -4685.197,E2 -4685.197} C_VEL
LIN {X 0,Y 523.743,Z 437.913,A -85,B 0,C 180,E1 -4685.969,E2 -4685.969} C_VEL
LIN {X 0,Y 523.959,Z 430.641,A -85,B 0,C 180,E1 -4686.669,E2 -4686.669} C_VEL
LIN {X 0,Y 524.002,Z 422.323,A -85,B 0,C 180,E1 -4687.282,E2 -4687.282} C_VEL
LIN {X 0,Y 524.185,Z 412.75,A -85,B 0,C 180,E1 -4687.802,E2 -4687.802} C_VEL
LIN {X 0,Y 523.451,Z 404.677,A -85,B 0,C 180,E1 -4688.153,E2 -4688.153} C_VEL
LIN {X 0,Y 523.517,Z 397.117,A -85,B 0,C 180,E1 -4691.479,E2 -4691.479} C_VEL
LIN {X 0,Y 523.654,Z 389.535,A -85,B 0,C 180,E1 -4694.912,E2 -4694.912} C_VEL
LIN {X 0,Y 523.735,Z 382.871,A -85,B 0,C 180,E1 -4697.977,E2 -4697.977} C_VEL
LIN {X 0,Y 523.788,Z 377.549,A -85,B 0,C 180,E1 -4700.418,E2 -4700.418} C_VEL
LIN {X 0,Y 523.888,Z 372.22,A -85,B 0,C 180,E1 -4702.895,E2 -4702.895} C_VEL
LIN {X 0,Y 524.055,Z 365.41,A -85,B 0,C 180,E1 -4706.035,E2 -4706.035} C_VEL
LIN {X 0,Y 524.145,Z 359.284,A -85,B 0,C 180,E1 -4708.862,E2 -4708.862} C_VEL
LIN {X 0,Y 524.024,Z 355.216,A -85,B 0,C 180,E1 -4710.794,E2 -4710.794} C_VEL
LIN {X 0,Y 523.937,Z 355.224,A -85,B 0,C 180,E1 -4714.29,E2 -4714.29} C_VEL
LIN {X 0,Y 523.911,Z 355.228,A -85,B 0,C 180,E1 -4717.132,E2 -4717.132} C_VEL
LIN {X 0,Y 523.972,Z 355.22,A -85,B 0,C 180,E1 -4720.134,E2 -4720.134} C_VEL
LIN {X 0,Y 523.929,Z 355.225,A -85,B 0,C 180,E1 -4723.166,E2 -4723.166} C_VEL
LIN {X 0,Y 523.945,Z 355.222,A -85,B 0,C 180,E1 -4725.772,E2 -4725.772} C_VEL
LIN {X 0,Y 523.945,Z 355.223,A -85,B 0,C 180,E1 -4728.908,E2 -4728.908} C_VEL
LIN {X 0,Y 523.918,Z 355.227,A -85,B 0,C 180,E1 -4731.898,E2 -4731.898} C_VEL
LIN {X 0,Y 523.928,Z 355.227,A -85,B 0,C 180,E1 -4734.911,E2 -4734.911} C_VEL
LIN {X 0,Y 523.942,Z 355.226,A -85,B 0,C 180,E1 -4737.679,E2 -4737.679} C_VEL
LIN {X 0,Y 523.925,Z 355.272,A -85,B 0,C 180,E1 -4738.886,E2 -4738.886} C_VEL
LIN {X 0,Y 526.104,Z 364.769,A -85,B 0,C 180,E1 -4741.255,E2 -4741.255} C_VEL
LIN {X 0,Y 526.377,Z 368.799,A -85,B 0,C 180,E1 -4742.14,E2 -4742.14} C_VEL
LIN {X 0,Y 525.559,Z 383.898,A -85,B 0,C 180,E1 -4745.13,E2 -4745.13} C_VEL
LIN {X 0,Y 524.987,Z 399.314,A -85,B 0,C 180,E1 -4747.986,E2 -4747.986} C_VEL
LIN {X 0,Y 524.655,Z 414.242,A -85,B 0,C 180,E1 -4750.638,E2 -4750.638} C_VEL
LIN {X 0,Y 524.329,Z 429.412,A -85,B 0,C 180,E1 -4753.251,E2 -4753.251} C_VEL
LIN {X 0,Y 524.041,Z 447.202,A -85,B 0,C 180,E1 -4756.228,E2 -4756.228} C_VEL
LIN {X 0,Y 524.041,Z 447.646,A -85,B 0,C 180,E1 -4756.303,E2 -4756.303} C_VEL
LIN {X 0,Y 525.329,Z 458.734,A -85,B 0,C 180,E1 -4756.534,E2 -4756.534} C_VEL
LIN {X 0,Y 525.157,Z 471.305,A -85,B 0,C 180,E1 -4756.899,E2 -4756.899} C_VEL
LIN {X 0,Y 524.937,Z 484.085,A -85,B 0,C 180,E1 -4757.434,E2 -4757.434} C_VEL
LIN {X 0,Y 524.674,Z 496.506,A -85,B 0,C 180,E1 -4758.128,E2 -4758.128} C_VEL
LIN {X 0,Y 524.383,Z 508.374,A -85,B 0,C 180,E1 -4758.99,E2 -4758.99} C_VEL
LIN {X 0,Y 524.075,Z 519.06,A -85,B 0,C 180,E1 -4759.96,E2 -4759.96} C_VEL
LIN {X 0,Y 523.874,Z 527.705,A -85,B 0,C 180,E1 -4760.93,E2 -4760.93} C_VEL
LIN {X 0,Y 523.688,Z 536.12,A -85,B 0,C 180,E1 -4762.093,E2 -4762.093} C_VEL
LIN {X 0,Y 523.575,Z 541.838,A -85,B 0,C 180,E1 -4763.061,E2 -4763.061} C_VEL
LIN {X 0,Y 523.544,Z 547.365,A -85,B 0,C 180,E1 -4764.222,E2 -4764.222} C_VEL
LIN {X 0,Y 523.361,Z 551.676,A -85,B 0,C 180,E1 -4765.378,E2 -4765.378} C_VEL
LIN {X 0,Y 523.443,Z 553.957,A -85,B 0,C 180,E1 -4766.151,E2 -4766.151} C_VEL
LIN {X 0,Y 523.367,Z 555.806,A -85,B 0,C 180,E1 -4766.921,E2 -4766.921} C_VEL
LIN {X 0,Y 523.335,Z 557.192,A -85,B 0,C 180,E1 -4767.691,E2 -4767.691} C_VEL
LIN {X 0,Y 523.25,Z 558.785,A -85,B 0,C 180,E1 -4769.23,E2 -4769.23} C_VEL
LIN {X 0,Y 523.246,Z 559,A -85,B 0,C 180,E1 -4770,E2 -4770} C_VEL
LIN {X 0,Y 523.275,Z 558.183,A -85,B 0,C 180,E1 -4771.539,E2 -4771.539} C_VEL
LIN {X 0,Y 523.335,Z 557.196,A -85,B 0,C 180,E1 -4772.309,E2 -4772.309} C_VEL
LIN {X 0,Y 523.367,Z 555.81,A -85,B 0,C 180,E1 -4773.079,E2 -4773.079} C_VEL
LIN {X 0,Y 523.441,Z 552.897,A -85,B 0,C 180,E1 -4774.235,E2 -4774.235} C_VEL
LIN {X 0,Y 523.464,Z 548.95,A -85,B 0,C 180,E1 -4775.393,E2 -4775.393} C_VEL
LIN {X 0,Y 523.519,Z 543.731,A -85,B 0,C 180,E1 -4776.577,E2 -4776.577} C_VEL
LIN {X 0,Y 523.665,Z 537.374,A -85,B 0,C 180,E1 -4777.713,E2 -4777.713} C_VEL
LIN {X 0,Y 523.845,Z 529.235,A -85,B 0,C 180,E1 -4778.875,E2 -4778.875} C_VEL
LIN {X 0,Y 524.033,Z 520.934,A -85,B 0,C 180,E1 -4779.846,E2 -4779.846} C_VEL
LIN {X 0,Y 524.342,Z 510.81,A -85,B 0,C 180,E1 -4780.815,E2 -4780.815} C_VEL
LIN {X 0,Y 524.573,Z 500.771,A -85,B 0,C 180,E1 -4781.593,E2 -4781.593} C_VEL
LIN {X 0,Y 524.846,Z 489.125,A -85,B 0,C 180,E1 -4782.313,E2 -4782.313} C_VEL
LIN {X 0,Y 525.072,Z 476.665,A -85,B 0,C 180,E1 -4782.906,E2 -4782.906} C_VEL
LIN {X 0,Y 525.285,Z 463.808,A -85,B 0,C 180,E1 -4783.344,E2 -4783.344} C_VEL
LIN {X 0,Y 525.187,Z 456.044,A -85,B 0,C 180,E1 -4783.534,E2 -4783.534} C_VEL
LIN {X 0,Y 524.042,Z 447.776,A -85,B 0,C 180,E1 -4783.722,E2 -4783.722} C_VEL
LIN {X 0,Y 524.345,Z 431.051,A -85,B 0,C 180,E1 -4786.548,E2 -4786.548} C_VEL
LIN {X 0,Y 524.661,Z 413.382,A -85,B 0,C 180,E1 -4789.565,E2 -4789.565} C_VEL
LIN {X 0,Y 525.019,Z 400.903,A -85,B 0,C 180,E1 -4791.806,E2 -4791.806} C_VEL
LIN {X 0,Y 525.585,Z 385.842,A -85,B 0,C 180,E1 -4794.594,E2 -4794.594} C_VEL
LIN {X 0,Y 526.183,Z 369.205,A -85,B 0,C 180,E1 -4797.655,E2 -4797.655} C_VEL
LIN {X 0,Y 526.132,Z 365.346,A -85,B 0,C 180,E1 -4798.403,E2 -4798.403} C_VEL
LIN {X 0,Y 523.943,Z 355.224,A -85,B 0,C 180,E1 -4800.589,E2 -4800.589} C_VEL
LIN {X 0,Y 523.961,Z 355.221,A -85,B 0,C 180,E1 -4803.734,E2 -4803.734} C_VEL
LIN {X 0,Y 523.905,Z 355.226,A -85,B 0,C 180,E1 -4806.401,E2 -4806.401} C_VEL
LIN {X 0,Y 523.921,Z 355.221,A -85,B 0,C 180,E1 -4809.085,E2 -4809.085} C_VEL
LIN {X 0,Y 523.958,Z 355.22,A -85,B 0,C 180,E1 -4812.118,E2 -4812.118} C_VEL
LIN {X 0,Y 523.958,Z 355.221,A -85,B 0,C 180,E1 -4815.308,E2 -4815.308} C_VEL
LIN {X 0,Y 523.96,Z 355.22,A -85,B 0,C 180,E1 -4818.689,E2 -4818.689} C_VEL
LIN {X 0,Y 523.919,Z 355.227,A -85,B 0,C 180,E1 -4821.898,E2 -4821.898} C_VEL
LIN {X 0,Y 523.937,Z 355.223,A -85,B 0,C 180,E1 -4824.909,E2 -4824.909} C_VEL
LIN {X 0,Y 523.937,Z 355.22,A -85,B 0,C 180,E1 -4827.68,E2 -4827.68} C_VEL
LIN {X 0,Y 523.956,Z 355.217,A -85,B 0,C 180,E1 -4830.676,E2 -4830.676} C_VEL
LIN {X 0,Y 523.977,Z 355.219,A -85,B 0,C 180,E1 -4833.729,E2 -4833.729} C_VEL
LIN {X 0,Y 523.927,Z 355.222,A -85,B 0,C 180,E1 -4836.27,E2 -4836.27} C_VEL
LIN {X 0,Y 523.948,Z 355.222,A -85,B 0,C 180,E1 -4838.767,E2 -4838.767} C_VEL
LIN {X 0,Y 523.952,Z 355.217,A -85,B 0,C 180,E1 -4841.221,E2 -4841.221} C_VEL
LIN {X 0,Y 523.94,Z 355.224,A -85,B 0,C 180,E1 -4843.639,E2 -4843.639} C_VEL
LIN {X 0,Y 523.948,Z 355.218,A -85,B 0,C 180,E1 -4846.028,E2 -4846.028} C_VEL
LIN {X 0,Y 524.014,Z 355.215,A -85,B 0,C 180,E1 -4848.394,E2 -4848.394} C_VEL
LIN {X 0,Y 524.005,Z 355.213,A -85,B 0,C 180,E1 -4851.516,E2 -4851.516} C_VEL
LIN {X 0,Y 524.084,Z 355.201,A -85,B 0,C 180,E1 -4854.614,E2 -4854.614} C_VEL
LIN {X 0,Y 524.112,Z 355.198,A -85,B 0,C 180,E1 -4857.694,E2 -4857.694} C_VEL
LIN {X 0,Y 524.126,Z 355.197,A -85,B 0,C 180,E1 -4860.768,E2 -4860.768} C_VEL
LIN {X 0,Y 524.073,Z 355.203,A -85,B 0,C 180,E1 -4863.075,E2 -4863.075} C_VEL
LIN {X 0,Y 524.048,Z 355.205,A -85,B 0,C 180,E1 -4866.159,E2 -4866.159} C_VEL
LIN {X 0,Y 524.002,Z 355.212,A -85,B 0,C 180,E1 -4869.262,E2 -4869.262} C_VEL
LIN {X 0,Y 524.027,Z 355.213,A -85,B 0,C 180,E1 -4871.751,E2 -4871.751} C_VEL
LIN {X 0,Y 523.995,Z 355.215,A -85,B 0,C 180,E1 -4875.052,E2 -4875.052} C_VEL
LIN {X 0,Y 523.966,Z 355.216,A -85,B 0,C 180,E1 -4877.969,E2 -4877.969} C_VEL
LIN {X 0,Y 523.974,Z 355.219,A -85,B 0,C 180,E1 -4880.41,E2 -4880.41} C_VEL
LIN {X 0,Y 523.919,Z 355.222,A -85,B 0,C 180,E1 -4882.893,E2 -4882.893} C_VEL
LIN {X 0,Y 523.955,Z 355.221,A -85,B 0,C 180,E1 -4885.419,E2 -4885.419} C_VEL
LIN {X 0,Y 523.969,Z 355.215,A -85,B 0,C 180,E1 -4887.999,E2 -4887.999} C_VEL
LIN {X 0,Y 523.946,Z 355.219,A -85,B 0,C 180,E1 -4890.855,E2 -4890.855} C_VEL
LIN {X 0,Y 523.963,Z 355.22,A -85,B 0,C 180,E1 -4893.735,E2 -4893.735} C_VEL
LIN {X 0,Y 523.921,Z 355.221,A -85,B 0,C 180,E1 -4896.404,E2 -4896.404} C_VEL
LIN {X 0,Y 523.924,Z 355.222,A -85,B 0,C 180,E1 -4899.085,E2 -4899.085} C_VEL
LIN {X 0,Y 523.959,Z 355.222,A -85,B 0,C 180,E1 -4902.119,E2 -4902.119} C_VEL
LIN {X 0,Y 523.958,Z 355.221,A -85,B 0,C 180,E1 -4905.309,E2 -4905.309} C_VEL
LIN {X 0,Y 523.925,Z 355.224,A -85,B 0,C 180,E1 -4906.911,E2 -4906.911} C_VEL
LIN {X 0,Y 523.257,Z 355.305,A -85,B 0,C 180,E1 -4907.553,E2 -4907.553} C_VEL
LIN {X 0,Y 520.413,Z 355.663,A -85,B 0,C 180,E1 -4908.594,E2 -4908.594} C_VEL
LIN {X 0,Y 518.007,Z 355.966,A -85,B 0,C 180,E1 -4909.433,E2 -4909.433} C_VEL
LIN {X 0,Y 516.97,Z 356.093,A -85,B 0,C 180,E1 -4910.081,E2 -4910.081} C_VEL
LIN {X 0,Y 516.883,Z 356.102,A -85,B 0,C 180,E1 -4910.3,E2 -4910.3} C_VEL
LIN {X 0,Y 516.879,Z 356.102,A -85,B 0,C 180,E1 -4913.343,E2 -4913.343} C_VEL
LIN {X 0,Y 516.91,Z 356.095,A -85,B 0,C 180,E1 -4916.121,E2 -4916.121} C_VEL
LIN {X 0,Y 516.893,Z 356.099,A -85,B 0,C 180,E1 -4918.936,E2 -4918.936} C_VEL
LIN {X 0,Y 516.922,Z 356.094,A -85,B 0,C 180,E1 -4921.585,E2 -4921.585} C_VEL
LIN {X 0,Y 516.934,Z 356.093,A -85,B 0,C 180,E1 -4924.211,E2 -4924.211} C_VEL
LIN {X 0,Y 516.868,Z 356.104,A -85,B 0,C 180,E1 -4926.776,E2 -4926.776} C_VEL
LIN {X 0,Y 516.942,Z 356.09,A -85,B 0,C 180,E1 -4929.732,E2 -4929.732} C_VEL
LIN {X 0,Y 516.933,Z 356.093,A -85,B 0,C 180,E1 -4932.596,E2 -4932.596} C_VEL
LIN {X 0,Y 516.946,Z 356.093,A -85,B 0,C 180,E1 -4935.03,E2 -4935.03} C_VEL
LIN {X 0,Y 516.969,Z 356.089,A -85,B 0,C 180,E1 -4938.234,E2 -4938.234} C_VEL
LIN {X 0,Y 516.971,Z 356.086,A -85,B 0,C 180,E1 -4941.4,E2 -4941.4} C_VEL
LIN {X 0,Y 517.006,Z 356.088,A -85,B 0,C 180,E1 -4943.757,E2 -4943.757} C_VEL
LIN {X 0,Y 517.015,Z 356.086,A -85,B 0,C 180,E1 -4946.883,E2 -4946.883} C_VEL
LIN {X 0,Y 517.089,Z 356.074,A -85,B 0,C 180,E1 -4950,E2 -4950} C_VEL
LIN {X 0,Y 517.015,Z 356.081,A -85,B 0,C 180,E1 -4953.117,E2 -4953.117} C_VEL
LIN {X 0,Y 517.006,Z 356.083,A -85,B 0,C 180,E1 -4956.243,E2 -4956.243} C_VEL
LIN {X 0,Y 516.956,Z 356.09,A -85,B 0,C 180,E1 -4959.389,E2 -4959.389} C_VEL
LIN {X 0,Y 516.957,Z 356.092,A -85,B 0,C 180,E1 -4961.808,E2 -4961.808} C_VEL
LIN {X 0,Y 516.949,Z 356.092,A -85,B 0,C 180,E1 -4965.147,E2 -4965.147} C_VEL
LIN {X 0,Y 516.928,Z 356.094,A -85,B 0,C 180,E1 -4968.222,E2 -4968.222} C_VEL
LIN {X 0,Y 516.916,Z 356.097,A -85,B 0,C 180,E1 -4970.702,E2 -4970.702} C_VEL
LIN {X 0,Y 516.895,Z 356.098,A -85,B 0,C 180,E1 -4974.073,E2 -4974.073} C_VEL
LIN {X 0,Y 516.93,Z 356.093,A -85,B 0,C 180,E1 -4976.658,E2 -4976.658} C_VEL
LIN {X 0,Y 516.915,Z 356.095,A -85,B 0,C 180,E1 -4979.524,E2 -4979.524} C_VEL
LIN {X 0,Y 516.901,Z 356.098,A -85,B 0,C 180,E1 -4982.544,E2 -4982.544} C_VEL
LIN {X 0,Y 516.87,Z 356.104,A -85,B 0,C 180,E1 -4985.33,E2 -4985.33} C_VEL
LIN {X 0,Y 516.884,Z 356.098,A -85,B 0,C 180,E1 -4987.943,E2 -4987.943} C_VEL
LIN {X 0,Y 516.888,Z 356.101,A -85,B 0,C 180,E1 -4990.742,E2 -4990.742} C_VEL
LIN {X 0,Y 516.908,Z 356.095,A -85,B 0,C 180,E1 -4992.829,E2 -4992.829} C_VEL
LIN {X 0,Y 516.885,Z 356.097,A -85,B 0,C 180,E1 -4996.107,E2 -4996.107} C_VEL
LIN {X 0,Y 516.917,Z 356.095,A -85,B 0,C 180,E1 -4998.399,E2 -4998.399} C_VEL
LIN {X 0,Y 516.886,Z 356.098,A -85,B 0,C 180,E1 -5001.284,E2 -5001.284} C_VEL
LIN {X 0,Y 516.892,Z 356.099,A -85,B 0,C 180,E1 -5004.221,E2 -5004.221} C_VEL
LIN {X 0,Y 516.899,Z 356.101,A -85,B 0,C 180,E1 -5007.053,E2 -5007.053} C_VEL
LIN {X 0,Y 517.024,Z 356.247,A -85,B 0,C 180,E1 -5010.009,E2 -5010.009} C_VEL
LIN {X 0,Y 516.811,Z 363.356,A -85,B 0,C 180,E1 -5013.336,E2 -5013.336} C_VEL
LIN {X 0,Y 516.776,Z 369.018,A -85,B 0,C 180,E1 -5015.921,E2 -5015.921} C_VEL
LIN {X 0,Y 516.623,Z 374.408,A -85,B 0,C 180,E1 -5018.451,E2 -5018.451} C_VEL
LIN {X 0,Y 516.555,Z 379.702,A -85,B 0,C 180,E1 -5020.941,E2 -5020.941} C_VEL
LIN {X 0,Y 516.455,Z 385.012,A -85,B 0,C 180,E1 -5023.395,E2 -5023.395} C_VEL
LIN {X 0,Y 516.416,Z 390.424,A -85,B 0,C 180,E1 -5025.82,E2 -5025.82} C_VEL
LIN {X 0,Y 516.374,Z 396.607,A -85,B 0,C 180,E1 -5028.506,E2 -5028.506} C_VEL
LIN {X 0,Y 516.313,Z 403.373,A -85,B 0,C 180,E1 -5031.389,E2 -5031.389} C_VEL
LIN {X 0,Y 516.344,Z 404.481,A -85,B 0,C 180,E1 -5031.857,E2 -5031.857} C_VEL
LIN {X 0,Y 517.139,Z 412.788,A -85,B 0,C 180,E1 -5032.189,E2 -5032.189} C_VEL
LIN {X 0,Y 516.994,Z 421.881,A -85,B 0,C 180,E1 -5032.678,E2 -5032.678} C_VEL
LIN {X 0,Y 516.872,Z 430.37,A -85,B 0,C 180,E1 -5033.297,E2 -5033.297} C_VEL
LIN {X 0,Y 516.664,Z 437.316,A -85,B 0,C 180,E1 -5033.949,E2 -5033.949} C_VEL
LIN {X 0,Y 516.625,Z 443.779,A -85,B 0,C 180,E1 -5034.731,E2 -5034.731} C_VEL
LIN {X 0,Y 516.546,Z 450.002,A -85,B 0,C 180,E1 -5035.708,E2 -5035.708} C_VEL
LIN {X 0,Y 516.546,Z 453.759,A -85,B 0,C 180,E1 -5036.49,E2 -5036.49} C_VEL
LIN {X 0,Y 516.317,Z 457.792,A -85,B 0,C 180,E1 -5037.66,E2 -5037.66} C_VEL
LIN {X 0,Y 516.256,Z 459.55,A -85,B 0,C 180,E1 -5038.44,E2 -5038.44} C_VEL
LIN {X 0,Y 516.24,Z 460.61,A -85,B 0,C 180,E1 -5039.22,E2 -5039.22} C_VEL
LIN {X 0,Y 516.24,Z 461.005,A -85,B 0,C 180,E1 -5040,E2 -5040} C_VEL
LIN {X 0,Y 516.244,Z 460.743,A -85,B 0,C 180,E1 -5040.78,E2 -5040.78} C_VEL
LIN {X 0,Y 516.265,Z 459.819,A -85,B 0,C 180,E1 -5041.56,E2 -5041.56} C_VEL
LIN {X 0,Y 516.423,Z 457.103,A -85,B 0,C 180,E1 -5042.73,E2 -5042.73} C_VEL
LIN {X 0,Y 516.543,Z 454.376,A -85,B 0,C 180,E1 -5043.51,E2 -5043.51} C_VEL
LIN {X 0,Y 516.562,Z 449.759,A -85,B 0,C 180,E1 -5044.487,E2 -5044.487} C_VEL
LIN {X 0,Y 516.659,Z 444.87,A -85,B 0,C 180,E1 -5045.268,E2 -5045.268} C_VEL
LIN {X 0,Y 516.736,Z 438.67,A -85,B 0,C 180,E1 -5046.051,E2 -5046.051} C_VEL
LIN {X 0,Y 516.97,Z 431.547,A -85,B 0,C 180,E1 -5046.751,E2 -5046.751} C_VEL
LIN {X 0,Y 517.023,Z 423.24,A -85,B 0,C 180,E1 -5047.38,E2 -5047.38} C_VEL
LIN {X 0,Y 517.202,Z 413.853,A -85,B 0,C 180,E1 -5047.908,E2 -5047.908} C_VEL
LIN {X 0,Y 516.681,Z 406.771,A -85,B 0,C 180,E1 -5048.211,E2 -5048.211} C_VEL
LIN {X 0,Y 516.427,Z 405.151,A -85,B 0,C 180,E1 -5048.289,E2 -5048.289} C_VEL
LIN {X 0,Y 516.489,Z 397.342,A -85,B 0,C 180,E1 -5051.777,E2 -5051.777} C_VEL
LIN {X 0,Y 516.62,Z 390.273,A -85,B 0,C 180,E1 -5055.011,E2 -5055.011} C_VEL
LIN {X 0,Y 516.696,Z 383.266,A -85,B 0,C 180,E1 -5058.231,E2 -5058.231} C_VEL
LIN {X 0,Y 516.785,Z 377.939,A -85,B 0,C 180,E1 -5060.707,E2 -5060.707} C_VEL
LIN {X 0,Y 516.887,Z 372.569,A -85,B 0,C 180,E1 -5063.223,E2 -5063.223} C_VEL
LIN {X 0,Y 517.065,Z 366.162,A -85,B 0,C 180,E1 -5066.223,E2 -5066.223} C_VEL
LIN {X 0,Y 517.205,Z 359.02,A -85,B 0,C 180,E1 -5069.581,E2 -5069.581} C_VEL
